LIN {X 0,Y 460.857,Z 363.08,A -85,B 0,C 180,E1 -7830,E2 -7830} C_VEL
LIN {X 0,Y 460.803,Z 363.083,A -85,B 0,C 180,E1 -7832.623,E2 -7832.623} C_VEL
LIN {X 0,Y 460.705,Z 363.097,A -85,B 0,C 180,E1 -7836.13,E2 -7836.13} C_VEL
LIN {X 0,Y 460.632,Z 363.107,A -85,B 0,C 180,E1 -7838.776,E2 -7838.776} C_VEL
LIN {X 0,Y 460.617,Z 363.108,A -85,B 0,C 180,E1 -7842.445,E2 -7842.445} C_VEL
LIN {X 0,Y 460.603,Z 363.11,A -85,B 0,C 180,E1 -7845.998,E2 -7845.998} C_VEL
LIN {X 0,Y 460.574,Z 363.115,A -85,B 0,C 180,E1 -7848.902,E2 -7848.902} C_VEL
LIN {X 0,Y 460.519,Z 363.121,A -85,B 0,C 180,E1 -7851.486,E2 -7851.486} C_VEL
LIN {X 0,Y 460.534,Z 363.116,A -85,B 0,C 180,E1 -7854.333,E2 -7854.333} C_VEL
LIN {X 0,Y 460.592,Z 363.111,A -85,B 0,C 180,E1 -7857.748,E2 -7857.748} C_VEL
LIN {X 0,Y 460.524,Z 363.12,A -85,B 0,C 180,E1 -7861.283,E2 -7861.283} C_VEL
LIN {X 0,Y 460.535,Z 363.117,A -85,B 0,C 180,E1 -7864.506,E2 -7864.506} C_VEL
LIN {X 0,Y 460.504,Z 363.122,A -85,B 0,C 180,E1 -7867.623,E2 -7867.623} C_VEL
LIN {X 0,Y 460.546,Z 363.118,A -85,B 0,C 180,E1 -7870.27,E2 -7870.27} C_VEL
LIN {X 0,Y 460.511,Z 363.123,A -85,B 0,C 180,E1 -7873.374,E2 -7873.374} C_VEL
LIN {X 0,Y 460.501,Z 363.121,A -85,B 0,C 180,E1 -7876.625,E2 -7876.625} C_VEL
LIN {X 0,Y 460.545,Z 363.117,A -85,B 0,C 180,E1 -7879.731,E2 -7879.731} C_VEL
LIN {X 0,Y 460.53,Z 363.121,A -85,B 0,C 180,E1 -7882.519,E2 -7882.519} C_VEL
LIN {X 0,Y 460.552,Z 363.117,A -85,B 0,C 180,E1 -7885.624,E2 -7885.624} C_VEL
LIN {X 0,Y 460.604,Z 363.114,A -85,B 0,C 180,E1 -7889.259,E2 -7889.259} C_VEL
LIN {X 0,Y 460.682,Z 363.307,A -85,B 0,C 180,E1 -7889.646,E2 -7889.646} C_VEL
LIN {X 0,Y 460.51,Z 369.483,A -85,B 0,C 180,E1 -7892.752,E2 -7892.752} C_VEL
LIN {X 0,Y 460.34,Z 375.322,A -85,B 0,C 180,E1 -7895.656,E2 -7895.656} C_VEL
LIN {X 0,Y 460.199,Z 381.499,A -85,B 0,C 180,E1 -7898.682,E2 -7898.682} C_VEL
LIN {X 0,Y 460.139,Z 386.881,A -85,B 0,C 180,E1 -7901.292,E2 -7901.292} C_VEL
LIN {X 0,Y 460.006,Z 394.526,A -85,B 0,C 180,E1 -7904.946,E2 -7904.946} C_VEL
LIN {X 0,Y 459.852,Z 402.194,A -85,B 0,C 180,E1 -7908.54,E2 -7908.54} C_VEL
LIN {X 0,Y 459.783,Z 406.743,A -85,B 0,C 180,E1 -7910.653,E2 -7910.653} C_VEL
LIN {X 0,Y 461.225,Z 417.498,A -85,B 0,C 180,E1 -7911.18,E2 -7911.18} C_VEL
LIN {X 0,Y 461.038,Z 426.889,A -85,B 0,C 180,E1 -7911.784,E2 -7911.784} C_VEL
LIN {X 0,Y 460.745,Z 435.524,A -85,B 0,C 180,E1 -7912.518,E2 -7912.518} C_VEL
LIN {X 0,Y 460.495,Z 443.706,A -85,B 0,C 180,E1 -7913.427,E2 -7913.427} C_VEL
LIN {X 0,Y 460.374,Z 451.186,A -85,B 0,C 180,E1 -7914.525,E2 -7914.525} C_VEL
LIN {X 0,Y 460.236,Z 456.815,A -85,B 0,C 180,E1 -7915.621,E2 -7915.621} C_VEL
LIN {X 0,Y 460.036,Z 461.668,A -85,B 0,C 180,E1 -7916.935,E2 -7916.935} C_VEL
LIN {X 0,Y 459.729,Z 464.779,A -85,B 0,C 180,E1 -7918.248,E2 -7918.248} C_VEL
LIN {X 0,Y 459.705,Z 465.955,A -85,B 0,C 180,E1 -7919.124,E2 -7919.124} C_VEL
LIN {X 0,Y 459.709,Z 466.457,A -85,B 0,C 180,E1 -7920,E2 -7920} C_VEL
LIN {X 0,Y 459.728,Z 466.292,A -85,B 0,C 180,E1 -7920.876,E2 -7920.876} C_VEL
LIN {X 0,Y 459.777,Z 465.459,A -85,B 0,C 180,E1 -7921.752,E2 -7921.752} C_VEL
LIN {X 0,Y 459.881,Z 463.94,A -85,B 0,C 180,E1 -7922.628,E2 -7922.628} C_VEL
LIN {X 0,Y 460.083,Z 461.69,A -85,B 0,C 180,E1 -7923.503,E2 -7923.503} C_VEL
LIN {X 0,Y 460.26,Z 458.652,A -85,B 0,C 180,E1 -7924.379,E2 -7924.379} C_VEL
LIN {X 0,Y 460.554,Z 453.616,A -85,B 0,C 180,E1 -7925.473,E2 -7925.473} C_VEL
LIN {X 0,Y 460.635,Z 448.398,A -85,B 0,C 180,E1 -7926.351,E2 -7926.351} C_VEL
LIN {X 0,Y 460.94,Z 441.818,A -85,B 0,C 180,E1 -7927.225,E2 -7927.225} C_VEL
LIN {X 0,Y 461.316,Z 433.586,A -85,B 0,C 180,E1 -7928.079,E2 -7928.079} C_VEL
LIN {X 0,Y 461.561,Z 425.177,A -85,B 0,C 180,E1 -7928.758,E2 -7928.758} C_VEL
LIN {X 0,Y 461.706,Z 418.277,A -85,B 0,C 180,E1 -7929.197,E2 -7929.197} C_VEL
LIN {X 0,Y 460.031,Z 408.765,A -85,B 0,C 180,E1 -7929.73,E2 -7929.73} C_VEL
LIN {X 0,Y 460.19,Z 403.416,A -85,B 0,C 180,E1 -7932.346,E2 -7932.346} C_VEL
LIN {X 0,Y 460.378,Z 396.222,A -85,B 0,C 180,E1 -7935.949,E2 -7935.949} C_VEL
LIN {X 0,Y 460.577,Z 390.465,A -85,B 0,C 180,E1 -7938.903,E2 -7938.903} C_VEL
LIN {X 0,Y 460.804,Z 383.745,A -85,B 0,C 180,E1 -7942.414,E2 -7942.414} C_VEL
LIN {X 0,Y 461.153,Z 377.222,A -85,B 0,C 180,E1 -7945.951,E2 -7945.951} C_VEL
LIN {X 0,Y 461.492,Z 371.525,A -85,B 0,C 180,E1 -7949.165,E2 -7949.165} C_VEL
LIN {X 0,Y 461.341,Z 367.729,A -85,B 0,C 180,E1 -7951.449,E2 -7951.449} C_VEL
LIN {X 0,Y 460.927,Z 364.949,A -85,B 0,C 180,E1 -7953.292,E2 -7953.292} C_VEL
LIN {X 0,Y 460.541,Z 363.122,A -85,B 0,C 180,E1 -7954.681,E2 -7954.681} C_VEL
LIN {X 0,Y 460.533,Z 363.122,A -85,B 0,C 180,E1 -7957.62,E2 -7957.62} C_VEL
LIN {X 0,Y 460.564,Z 363.118,A -85,B 0,C 180,E1 -7960.272,E2 -7960.272} C_VEL
LIN {X 0,Y 460.528,Z 363.122,A -85,B 0,C 180,E1 -7963.372,E2 -7963.372} C_VEL
LIN {X 0,Y 460.512,Z 363.124,A -85,B 0,C 180,E1 -7966.626,E2 -7966.626} C_VEL
LIN {X 0,Y 460.546,Z 363.121,A -85,B 0,C 180,E1 -7969.73,E2 -7969.73} C_VEL
LIN {X 0,Y 460.502,Z 363.126,A -85,B 0,C 180,E1 -7972.524,E2 -7972.524} C_VEL
LIN {X 0,Y 460.517,Z 363.332,A -85,B 0,C 180,E1 -7973.621,E2 -7973.621} C_VEL
LIN {X 0,Y 461.719,Z 367.784,A -85,B 0,C 180,E1 -7975.723,E2 -7975.723} C_VEL
LIN {X 0,Y 463.014,Z 373.479,A -85,B 0,C 180,E1 -7977.909,E2 -7977.909} C_VEL
LIN {X 0,Y 464.367,Z 379.853,A -85,B 0,C 180,E1 -7980.037,E2 -7980.037} C_VEL
LIN {X 0,Y 464.726,Z 384.238,A -85,B 0,C 180,E1 -7981.298,E2 -7981.298} C_VEL
LIN {X 0,Y 463.505,Z 394.628,A -85,B 0,C 180,E1 -7983.914,E2 -7983.914} C_VEL
LIN {X 0,Y 462.368,Z 407.715,A -85,B 0,C 180,E1 -7986.958,E2 -7986.958} C_VEL
LIN {X 0,Y 461.482,Z 422.533,A -85,B 0,C 180,E1 -7990.193,E2 -7990.193} C_VEL
LIN {X 0,Y 460.787,Z 438.027,A -85,B 0,C 180,E1 -7993.405,E2 -7993.405} C_VEL
LIN {X 0,Y 460.585,Z 444.606,A -85,B 0,C 180,E1 -7994.739,E2 -7994.739} C_VEL
LIN {X 0,Y 462.033,Z 459.219,A -85,B 0,C 180,E1 -7995.154,E2 -7995.154} C_VEL
LIN {X 0,Y 462.409,Z 464.775,A -85,B 0,C 180,E1 -7995.364,E2 -7995.364} C_VEL
LIN {X 0,Y 462.099,Z 476.978,A -85,B 0,C 180,E1 -7995.916,E2 -7995.916} C_VEL
LIN {X 0,Y 461.61,Z 489.57,A -85,B 0,C 180,E1 -7996.686,E2 -7996.686} C_VEL
LIN {X 0,Y 461.252,Z 500.147,A -85,B 0,C 180,E1 -7997.513,E2 -7997.513} C_VEL
LIN {X 0,Y 460.68,Z 509.899,A -85,B 0,C 180,E1 -7998.449,E2 -7998.449} C_VEL
LIN {X 0,Y 460.444,Z 518.389,A -85,B 0,C 180,E1 -7999.446,E2 -7999.446} C_VEL
LIN {X 0,Y 460.109,Z 527.598,A -85,B 0,C 180,E1 -8000.771,E2 -8000.771} C_VEL
LIN {X 0,Y 459.907,Z 535.009,A -85,B 0,C 180,E1 -8002.095,E2 -8002.095} C_VEL
LIN {X 0,Y 459.813,Z 541.057,A -85,B 0,C 180,E1 -8003.461,E2 -8003.461} C_VEL
LIN {X 0,Y 459.737,Z 545.498,A -85,B 0,C 180,E1 -8004.737,E2 -8004.737} C_VEL
LIN {X 0,Y 459.701,Z 547.925,A -85,B 0,C 180,E1 -8005.616,E2 -8005.616} C_VEL
LIN {X 0,Y 459.75,Z 549.915,A -85,B 0,C 180,E1 -8006.494,E2 -8006.494} C_VEL
LIN {X 0,Y 459.762,Z 551.424,A -85,B 0,C 180,E1 -8007.371,E2 -8007.371} C_VEL
LIN {X 0,Y 459.603,Z 553.141,A -85,B 0,C 180,E1 -8009.124,E2 -8009.124} C_VEL
LIN {X 0,Y 459.605,Z 553.392,A -85,B 0,C 180,E1 -8010,E2 -8010} C_VEL
LIN {X 0,Y 459.6,Z 553.186,A -85,B 0,C 180,E1 -8010.876,E2 -8010.876} C_VEL
LIN {X 0,Y 459.762,Z 551.579,A -85,B 0,C 180,E1 -8012.628,E2 -8012.628} C_VEL
LIN {X 0,Y 459.745,Z 550.107,A -85,B 0,C 180,E1 -8013.505,E2 -8013.505} C_VEL
LIN {X 0,Y 459.657,Z 547.047,A -85,B 0,C 180,E1 -8014.824,E2 -8014.824} C_VEL
LIN {X 0,Y 459.729,Z 542.895,A -85,B 0,C 180,E1 -8016.143,E2 -8016.143} C_VEL
LIN {X 0,Y 459.854,Z 537.524,A -85,B 0,C 180,E1 -8017.464,E2 -8017.464} C_VEL
LIN {X 0,Y 460.017,Z 530.749,A -85,B 0,C 180,E1 -8018.788,E2 -8018.788} C_VEL
LIN {X 0,Y 460.304,Z 522.289,A -85,B 0,C 180,E1 -8020.112,E2 -8020.112} C_VEL
LIN {X 0,Y 460.715,Z 513.529,A -85,B 0,C 180,E1 -8021.215,E2 -8021.215} C_VEL
LIN {X 0,Y 461.128,Z 503.892,A -85,B 0,C 180,E1 -8022.208,E2 -8022.208} C_VEL
LIN {X 0,Y 461.557,Z 493.026,A -85,B 0,C 180,E1 -8023.116,E2 -8023.116} C_VEL
LIN {X 0,Y 461.969,Z 481.615,A -85,B 0,C 180,E1 -8023.863,E2 -8023.863} C_VEL
LIN {X 0,Y 462.419,Z 468.145,A -85,B 0,C 180,E1 -8024.523,E2 -8024.523} C_VEL
LIN {X 0,Y 462.274,Z 461.426,A -85,B 0,C 180,E1 -8024.781,E2 -8024.781} C_VEL
LIN {X 0,Y 461.043,Z 449.191,A -85,B 0,C 180,E1 -8025.143,E2 -8025.143} C_VEL
LIN {X 0,Y 460.644,Z 445.197,A -85,B 0,C 180,E1 -8025.259,E2 -8025.259} C_VEL
LIN {X 0,Y 461.241,Z 428.609,A -85,B 0,C 180,E1 -8028.662,E2 -8028.662} C_VEL
LIN {X 0,Y 462.088,Z 413.087,A -85,B 0,C 180,E1 -8031.911,E2 -8031.911} C_VEL
LIN {X 0,Y 463.079,Z 396.786,A -85,B 0,C 180,E1 -8035.388,E2 -8035.388} C_VEL
LIN {X 0,Y 464.179,Z 382.26,A -85,B 0,C 180,E1 -8038.578,E2 -8038.578} C_VEL
LIN {X 0,Y 463.806,Z 378.299,A -85,B 0,C 180,E1 -8039.503,E2 -8039.503} C_VEL
LIN {X 0,Y 461.42,Z 367.379,A -85,B 0,C 180,E1 -8042.215,E2 -8042.215} C_VEL
LIN {X 0,Y 460.595,Z 363.115,A -85,B 0,C 180,E1 -8043.319,E2 -8043.319} C_VEL
LIN {X 0,Y 460.478,Z 363.127,A -85,B 0,C 180,E1 -8046.529,E2 -8046.529} C_VEL
LIN {X 0,Y 460.534,Z 363.12,A -85,B 0,C 180,E1 -8049.862,E2 -8049.862} C_VEL
LIN {X 0,Y 460.518,Z 363.121,A -85,B 0,C 180,E1 -8052.901,E2 -8052.901} C_VEL
LIN {X 0,Y 460.521,Z 363.121,A -85,B 0,C 180,E1 -8055.829,E2 -8055.829} C_VEL
LIN {X 0,Y 460.535,Z 363.117,A -85,B 0,C 180,E1 -8058.989,E2 -8058.989} C_VEL
LIN {X 0,Y 460.528,Z 363.118,A -85,B 0,C 180,E1 -8061.267,E2 -8061.267} C_VEL
LIN {X 0,Y 460.514,Z 363.121,A -85,B 0,C 180,E1 -8064.555,E2 -8064.555} C_VEL
LIN {X 0,Y 460.532,Z 363.119,A -85,B 0,C 180,E1 -8067.716,E2 -8067.716} C_VEL
LIN {X 0,Y 460.541,Z 363.116,A -85,B 0,C 180,E1 -8070.769,E2 -8070.769} C_VEL
LIN {X 0,Y 460.564,Z 363.118,A -85,B 0,C 180,E1 -8073.735,E2 -8073.735} C_VEL
LIN {X 0,Y 460.547,Z 363.119,A -85,B 0,C 180,E1 -8076.624,E2 -8076.624} C_VEL
LIN {X 0,Y 460.553,Z 363.116,A -85,B 0,C 180,E1 -8079.453,E2 -8079.453} C_VEL
LIN {X 0,Y 460.561,Z 363.115,A -85,B 0,C 180,E1 -8082.23,E2 -8082.23} C_VEL
LIN {X 0,Y 460.569,Z 363.114,A -85,B 0,C 180,E1 -8084.965,E2 -8084.965} C_VEL
LIN {X 0,Y 460.613,Z 363.11,A -85,B 0,C 180,E1 -8088.559,E2 -8088.559} C_VEL
LIN {X 0,Y 460.696,Z 363.099,A -85,B 0,C 180,E1 -8092.109,E2 -8092.109} C_VEL
LIN {X 0,Y 460.698,Z 363.097,A -85,B 0,C 180,E1 -8094.748,E2 -8094.748} C_VEL
LIN {X 0,Y 460.826,Z 363.083,A -85,B 0,C 180,E1 -8097.378,E2 -8097.378} C_VEL
LIN {X 0,Y 460.855,Z 363.081,A -85,B 0,C 180,E1 -8100,E2 -8100} C_VEL
LIN {X 0,Y 460.802,Z 363.084,A -85,B 0,C 180,E1 -8102.623,E2 -8102.623} C_VEL
LIN {X 0,Y 460.711,Z 363.095,A -85,B 0,C 180,E1 -8106.13,E2 -8106.13} C_VEL
LIN {X 0,Y 460.631,Z 363.109,A -85,B 0,C 180,E1 -8108.776,E2 -8108.776} C_VEL
LIN {X 0,Y 460.636,Z 363.106,A -85,B 0,C 180,E1 -8112.457,E2 -8112.457} C_VEL
LIN {X 0,Y 460.601,Z 363.108,A -85,B 0,C 180,E1 -8115.998,E2 -8115.998} C_VEL
LIN {X 0,Y 460.573,Z 363.116,A -85,B 0,C 180,E1 -8118.902,E2 -8118.902} C_VEL
LIN {X 0,Y 460.517,Z 363.122,A -85,B 0,C 180,E1 -8121.486,E2 -8121.486} C_VEL
LIN {X 0,Y 460.544,Z 363.116,A -85,B 0,C 180,E1 -8124.332,E2 -8124.332} C_VEL
LIN {X 0,Y 460.574,Z 363.115,A -85,B 0,C 180,E1 -8127.244,E2 -8127.244} C_VEL
LIN {X 0,Y 460.512,Z 363.122,A -85,B 0,C 180,E1 -8130.24,E2 -8130.24} C_VEL
LIN {X 0,Y 460.53,Z 363.122,A -85,B 0,C 180,E1 -8133.325,E2 -8133.325} C_VEL
LIN {X 0,Y 460.48,Z 363.125,A -85,B 0,C 180,E1 -8136.529,E2 -8136.529} C_VEL
LIN {X 0,Y 460.546,Z 363.119,A -85,B 0,C 180,E1 -8138.898,E2 -8138.898} C_VEL
LIN {X 0,Y 460.524,Z 363.122,A -85,B 0,C 180,E1 -8142.182,E2 -8142.182} C_VEL
LIN {X 0,Y 460.522,Z 363.121,A -85,B 0,C 180,E1 -8145.412,E2 -8145.412} C_VEL
LIN {X 0,Y 460.537,Z 363.119,A -85,B 0,C 180,E1 -8148.397,E2 -8148.397} C_VEL
LIN {X 0,Y 460.528,Z 363.119,A -85,B 0,C 180,E1 -8151.267,E2 -8151.267} C_VEL
LIN {X 0,Y 460.512,Z 363.122,A -85,B 0,C 180,E1 -8154.555,E2 -8154.555} C_VEL
LIN {X 0,Y 460.533,Z 363.118,A -85,B 0,C 180,E1 -8157.716,E2 -8157.716} C_VEL
LIN {X 0,Y 460.542,Z 363.118,A -85,B 0,C 180,E1 -8160.769,E2 -8160.769} C_VEL
LIN {X 0,Y 460.565,Z 363.116,A -85,B 0,C 180,E1 -8163.735,E2 -8163.735} C_VEL
LIN {X 0,Y 460.548,Z 363.119,A -85,B 0,C 180,E1 -8166.624,E2 -8166.624} C_VEL
LIN {X 0,Y 460.555,Z 363.114,A -85,B 0,C 180,E1 -8169.453,E2 -8169.453} C_VEL
LIN {X 0,Y 460.563,Z 363.118,A -85,B 0,C 180,E1 -8172.23,E2 -8172.23} C_VEL
LIN {X 0,Y 460.573,Z 363.115,A -85,B 0,C 180,E1 -8174.965,E2 -8174.965} C_VEL
LIN {X 0,Y 460.614,Z 363.112,A -85,B 0,C 180,E1 -8178.56,E2 -8178.56} C_VEL
LIN {X 0,Y 460.58,Z 363.112,A -85,B 0,C 180,E1 -8179.225,E2 -8179.225} C_VEL
LIN {X 0,Y 459.924,Z 363.197,A -85,B 0,C 180,E1 -8179.955,E2 -8179.955} C_VEL
LIN {X 0,Y 457.104,Z 363.545,A -85,B 0,C 180,E1 -8181.141,E2 -8181.141} C_VEL
LIN {X 0,Y 454.722,Z 363.846,A -85,B 0,C 180,E1 -8182.098,E2 -8182.098} C_VEL
LIN {X 0,Y 453.709,Z 363.968,A -85,B 0,C 180,E1 -8182.837,E2 -8182.837} C_VEL
LIN {X 0,Y 453.632,Z 363.977,A -85,B 0,C 180,E1 -8183.087,E2 -8183.087} C_VEL
LIN {X 0,Y 453.672,Z 363.973,A -85,B 0,C 180,E1 -8184.667,E2 -8184.667} C_VEL
LIN {X 0,Y 453.747,Z 363.965,A -85,B 0,C 180,E1 -8187.337,E2 -8187.337} C_VEL
LIN {X 0,Y 453.828,Z 363.955,A -85,B 0,C 180,E1 -8190,E2 -8190} C_VEL
LIN {X 0,Y 453.747,Z 363.962,A -85,B 0,C 180,E1 -8192.663,E2 -8192.663} C_VEL
LIN {X 0,Y 453.673,Z 363.973,A -85,B 0,C 180,E1 -8196.226,E2 -8196.226} C_VEL
LIN {X 0,Y 453.596,Z 363.984,A -85,B 0,C 180,E1 -8198.913,E2 -8198.913} C_VEL
LIN {X 0,Y 453.567,Z 363.985,A -85,B 0,C 180,E1 -8202.529,E2 -8202.529} C_VEL
LIN {X 0,Y 453.548,Z 363.988,A -85,B 0,C 180,E1 -8206.196,E2 -8206.196} C_VEL
LIN {X 0,Y 453.524,Z 363.994,A -85,B 0,C 180,E1 -8209.041,E2 -8209.041} C_VEL
LIN {X 0,Y 453.48,Z 364,A -85,B 0,C 180,E1 -8211.836,E2 -8211.836} C_VEL
LIN {X 0,Y 453.504,Z 363.992,A -85,B 0,C 180,E1 -8214.735,E2 -8214.735} C_VEL
LIN {X 0,Y 453.541,Z 363.99,A -85,B 0,C 180,E1 -8217.961,E2 -8217.961} C_VEL
LIN {X 0,Y 453.469,Z 363.999,A -85,B 0,C 180,E1 -8221.525,E2 -8221.525} C_VEL
LIN {X 0,Y 453.49,Z 363.995,A -85,B 0,C 180,E1 -8224.777,E2 -8224.777} C_VEL
LIN {X 0,Y 453.468,Z 363.999,A -85,B 0,C 180,E1 -8228.312,E2 -8228.312} C_VEL
LIN {X 0,Y 453.497,Z 363.996,A -85,B 0,C 180,E1 -8230.609,E2 -8230.609} C_VEL
LIN {X 0,Y 453.465,Z 364,A -85,B 0,C 180,E1 -8233.245,E2 -8233.245} C_VEL
LIN {X 0,Y 453.466,Z 363.999,A -85,B 0,C 180,E1 -8235.779,E2 -8235.779} C_VEL
LIN {X 0,Y 453.482,Z 363.996,A -85,B 0,C 180,E1 -8238.209,E2 -8238.209} C_VEL
LIN {X 0,Y 453.513,Z 363.996,A -85,B 0,C 180,E1 -8240.791,E2 -8240.791} C_VEL
LIN {X 0,Y 453.46,Z 364,A -85,B 0,C 180,E1 -8243.917,E2 -8243.917} C_VEL
LIN {X 0,Y 453.487,Z 364,A -85,B 0,C 180,E1 -8247.151,E2 -8247.151} C_VEL
LIN {X 0,Y 453.577,Z 364.027,A -85,B 0,C 180,E1 -8249.503,E2 -8249.503} C_VEL
LIN {X 0,Y 453.506,Z 369.486,A -85,B 0,C 180,E1 -8252.295,E2 -8252.295} C_VEL
LIN {X 0,Y 453.315,Z 375.395,A -85,B 0,C 180,E1 -8255.254,E2 -8255.254} C_VEL
LIN {X 0,Y 453.165,Z 381.948,A -85,B 0,C 180,E1 -8258.517,E2 -8258.517} C_VEL
LIN {X 0,Y 453.027,Z 388.938,A -85,B 0,C 180,E1 -8261.924,E2 -8261.924} C_VEL
LIN {X 0,Y 452.966,Z 394.742,A -85,B 0,C 180,E1 -8264.706,E2 -8264.706} C_VEL
LIN {X 0,Y 452.795,Z 402.443,A -85,B 0,C 180,E1 -8268.359,E2 -8268.359} C_VEL
LIN {X 0,Y 452.734,Z 407.048,A -85,B 0,C 180,E1 -8270.506,E2 -8270.506} C_VEL
LIN {X 0,Y 454.161,Z 416.831,A -85,B 0,C 180,E1 -8270.986,E2 -8270.986} C_VEL
LIN {X 0,Y 454.065,Z 425.727,A -85,B 0,C 180,E1 -8271.544,E2 -8271.544} C_VEL
LIN {X 0,Y 453.838,Z 433.911,A -85,B 0,C 180,E1 -8272.213,E2 -8272.213} C_VEL
LIN {X 0,Y 453.47,Z 442.344,A -85,B 0,C 180,E1 -8273.101,E2 -8273.101} C_VEL
LIN {X 0,Y 453.405,Z 448.927,A -85,B 0,C 180,E1 -8273.994,E2 -8273.994} C_VEL
LIN {X 0,Y 453.237,Z 455.281,A -85,B 0,C 180,E1 -8275.108,E2 -8275.108} C_VEL
LIN {X 0,Y 453.022,Z 460.828,A -85,B 0,C 180,E1 -8276.442,E2 -8276.442} C_VEL
LIN {X 0,Y 452.8,Z 463.498,A -85,B 0,C 180,E1 -8277.331,E2 -8277.331} C_VEL
LIN {X 0,Y 452.666,Z 465.412,A -85,B 0,C 180,E1 -8278.221,E2 -8278.221} C_VEL
LIN {X 0,Y 452.637,Z 466.617,A -85,B 0,C 180,E1 -8279.11,E2 -8279.11} C_VEL
LIN {X 0,Y 452.643,Z 467.146,A -85,B 0,C 180,E1 -8280,E2 -8280} C_VEL
LIN {X 0,Y 452.666,Z 467.006,A -85,B 0,C 180,E1 -8280.89,E2 -8280.89} C_VEL
LIN {X 0,Y 452.719,Z 466.196,A -85,B 0,C 180,E1 -8281.779,E2 -8281.779} C_VEL
LIN {X 0,Y 452.83,Z 464.701,A -85,B 0,C 180,E1 -8282.669,E2 -8282.669} C_VEL
LIN {X 0,Y 453.048,Z 462.476,A -85,B 0,C 180,E1 -8283.558,E2 -8283.558} C_VEL
LIN {X 0,Y 453.237,Z 459.477,A -85,B 0,C 180,E1 -8284.447,E2 -8284.447} C_VEL
LIN {X 0,Y 453.547,Z 454.511,A -85,B 0,C 180,E1 -8285.558,E2 -8285.558} C_VEL
LIN {X 0,Y 453.728,Z 447.9,A -85,B 0,C 180,E1 -8286.671,E2 -8286.671} C_VEL
LIN {X 0,Y 454.14,Z 440.066,A -85,B 0,C 180,E1 -8287.668,E2 -8287.668} C_VEL
LIN {X 0,Y 454.448,Z 432.198,A -85,B 0,C 180,E1 -8288.448,E2 -8288.448} C_VEL
LIN {X 0,Y 454.75,Z 423.545,A -85,B 0,C 180,E1 -8289.115,E2 -8289.115} C_VEL
LIN {X 0,Y 454.682,Z 418.192,A -85,B 0,C 180,E1 -8289.453,E2 -8289.453} C_VEL
LIN {X 0,Y 453.006,Z 409.211,A -85,B 0,C 180,E1 -8289.967,E2 -8289.967} C_VEL
LIN {X 0,Y 453.164,Z 404.055,A -85,B 0,C 180,E1 -8292.54,E2 -8292.54} C_VEL
LIN {X 0,Y 453.392,Z 396.849,A -85,B 0,C 180,E1 -8296.202,E2 -8296.202} C_VEL
LIN {X 0,Y 453.572,Z 391.35,A -85,B 0,C 180,E1 -8299.058,E2 -8299.058} C_VEL
LIN {X 0,Y 453.768,Z 386.166,A -85,B 0,C 180,E1 -8301.821,E2 -8301.821} C_VEL
LIN {X 0,Y 454.027,Z 380.917,A -85,B 0,C 180,E1 -8304.705,E2 -8304.705} C_VEL
LIN {X 0,Y 454.4,Z 375.73,A -85,B 0,C 180,E1 -8307.645,E2 -8307.645} C_VEL
LIN {X 0,Y 454.627,Z 371.692,A -85,B 0,C 180,E1 -8310.037,E2 -8310.037} C_VEL
LIN {X 0,Y 454.186,Z 367.518,A -85,B 0,C 180,E1 -8312.792,E2 -8312.792} C_VEL
LIN {X 0,Y 453.479,Z 364.001,A -85,B 0,C 180,E1 -8315.465,E2 -8315.465} C_VEL
LIN {X 0,Y 453.489,Z 364,A -85,B 0,C 180,E1 -8318.309,E2 -8318.309} C_VEL
LIN {X 0,Y 453.519,Z 363.995,A -85,B 0,C 180,E1 -8320.606,E2 -8320.606} C_VEL
LIN {X 0,Y 453.485,Z 363.999,A -85,B 0,C 180,E1 -8323.248,E2 -8323.248} C_VEL
LIN {X 0,Y 453.476,Z 364,A -85,B 0,C 180,E1 -8325.78,E2 -8325.78} C_VEL
LIN {X 0,Y 453.485,Z 364,A -85,B 0,C 180,E1 -8328.21,E2 -8328.21} C_VEL
LIN {X 0,Y 453.513,Z 363.996,A -85,B 0,C 180,E1 -8330.791,E2 -8330.791} C_VEL
LIN {X 0,Y 453.488,Z 364.196,A -85,B 0,C 180,E1 -8332.668,E2 -8332.668} C_VEL
LIN {X 0,Y 454.704,Z 368.932,A -85,B 0,C 180,E1 -8335.118,E2 -8335.118} C_VEL
LIN {X 0,Y 456.017,Z 374.334,A -85,B 0,C 180,E1 -8337.356,E2 -8337.356} C_VEL
LIN {X 0,Y 457.641,Z 382.209,A -85,B 0,C 180,E1 -8340.059,E2 -8340.059} C_VEL
LIN {X 0,Y 457.921,Z 385.915,A -85,B 0,C 180,E1 -8341.168,E2 -8341.168} C_VEL
LIN {X 0,Y 456.749,Z 394.867,A -85,B 0,C 180,E1 -8343.498,E2 -8343.498} C_VEL
LIN {X 0,Y 455.483,Z 407.713,A -85,B 0,C 180,E1 -8346.589,E2 -8346.589} C_VEL
LIN {X 0,Y 454.554,Z 422.357,A -85,B 0,C 180,E1 -8349.878,E2 -8349.878} C_VEL
LIN {X 0,Y 453.777,Z 437.577,A -85,B 0,C 180,E1 -8353.118,E2 -8353.118} C_VEL
LIN {X 0,Y 453.57,Z 444.565,A -85,B 0,C 180,E1 -8354.52,E2 -8354.52} C_VEL
LIN {X 0,Y 454.846,Z 457.367,A -85,B 0,C 180,E1 -8354.886,E2 -8354.886} C_VEL
LIN {X 0,Y 455.465,Z 465.322,A -85,B 0,C 180,E1 -8355.193,E2 -8355.193} C_VEL
LIN {X 0,Y 455.152,Z 476.153,A -85,B 0,C 180,E1 -8355.696,E2 -8355.696} C_VEL
LIN {X 0,Y 454.648,Z 488.774,A -85,B 0,C 180,E1 -8356.479,E2 -8356.479} C_VEL
LIN {X 0,Y 454.225,Z 500.002,A -85,B 0,C 180,E1 -8357.372,E2 -8357.372} C_VEL
LIN {X 0,Y 453.607,Z 510.137,A -85,B 0,C 180,E1 -8358.38,E2 -8358.38} C_VEL
LIN {X 0,Y 453.317,Z 519.313,A -85,B 0,C 180,E1 -8359.504,E2 -8359.504} C_VEL
LIN {X 0,Y 453.015,Z 528.254,A -85,B 0,C 180,E1 -8360.85,E2 -8360.85} C_VEL
LIN {X 0,Y 452.815,Z 535.355,A -85,B 0,C 180,E1 -8362.195,E2 -8362.195} C_VEL
LIN {X 0,Y 452.731,Z 540.774,A -85,B 0,C 180,E1 -8363.469,E2 -8363.469} C_VEL
LIN {X 0,Y 452.677,Z 544.812,A -85,B 0,C 180,E1 -8364.655,E2 -8364.655} C_VEL
LIN {X 0,Y 452.65,Z 548.3,A -85,B 0,C 180,E1 -8365.993,E2 -8365.993} C_VEL
LIN {X 0,Y 452.707,Z 550.755,A -85,B 0,C 180,E1 -8367.33,E2 -8367.33} C_VEL
LIN {X 0,Y 452.536,Z 552.476,A -85,B 0,C 180,E1 -8369.11,E2 -8369.11} C_VEL
LIN {X 0,Y 452.536,Z 552.725,A -85,B 0,C 180,E1 -8370,E2 -8370} C_VEL
LIN {X 0,Y 452.59,Z 551.909,A -85,B 0,C 180,E1 -8371.78,E2 -8371.78} C_VEL
LIN {X 0,Y 452.706,Z 550.904,A -85,B 0,C 180,E1 -8372.669,E2 -8372.669} C_VEL
LIN {X 0,Y 452.674,Z 549.416,A -85,B 0,C 180,E1 -8373.56,E2 -8373.56} C_VEL
LIN {X 0,Y 452.589,Z 546.337,A -85,B 0,C 180,E1 -8374.899,E2 -8374.899} C_VEL
LIN {X 0,Y 452.691,Z 541.261,A -85,B 0,C 180,E1 -8376.486,E2 -8376.486} C_VEL
LIN {X 0,Y 452.837,Z 534.667,A -85,B 0,C 180,E1 -8378.029,E2 -8378.029} C_VEL
LIN {X 0,Y 453.044,Z 527.293,A -85,B 0,C 180,E1 -8379.374,E2 -8379.374} C_VEL
LIN {X 0,Y 453.443,Z 518.107,A -85,B 0,C 180,E1 -8380.719,E2 -8380.719} C_VEL
LIN {X 0,Y 453.872,Z 507.418,A -85,B 0,C 180,E1 -8381.953,E2 -8381.953} C_VEL
LIN {X 0,Y 454.33,Z 496.566,A -85,B 0,C 180,E1 -8382.955,E2 -8382.955} C_VEL
LIN {X 0,Y 454.815,Z 485.74,A -85,B 0,C 180,E1 -8383.744,E2 -8383.744} C_VEL
LIN {X 0,Y 455.293,Z 472.8,A -85,B 0,C 180,E1 -8384.47,E2 -8384.47} C_VEL
LIN {X 0,Y 455.356,Z 462.669,A -85,B 0,C 180,E1 -8384.896,E2 -8384.896} C_VEL
LIN {X 0,Y 454.237,Z 450.854,A -85,B 0,C 180,E1 -8385.278,E2 -8385.278} C_VEL
LIN {X 0,Y 453.578,Z 444.953,A -85,B 0,C 180,E1 -8385.441,E2 -8385.441} C_VEL
LIN {X 0,Y 454.196,Z 429.258,A -85,B 0,C 180,E1 -8388.728,E2 -8388.728} C_VEL
LIN {X 0,Y 455.014,Z 415.009,A -85,B 0,C 180,E1 -8391.758,E2 -8391.758} C_VEL
LIN {X 0,Y 456.077,Z 398.702,A -85,B 0,C 180,E1 -8395.316,E2 -8395.316} C_VEL
LIN {X 0,Y 457.183,Z 384.551,A -85,B 0,C 180,E1 -8398.46,E2 -8398.46} C_VEL
LIN {X 0,Y 457.263,Z 381.851,A -85,B 0,C 180,E1 -8399.083,E2 -8399.083} C_VEL
LIN {X 0,Y 454.968,Z 370.857,A -85,B 0,C 180,E1 -8401.832,E2 -8401.832} C_VEL
LIN {X 0,Y 453.521,Z 363.995,A -85,B 0,C 180,E1 -8403.62,E2 -8403.62} C_VEL
LIN {X 0,Y 453.453,Z 364.001,A -85,B 0,C 180,E1 -8407.189,E2 -8407.189} C_VEL
LIN {X 0,Y 453.491,Z 363.995,A -85,B 0,C 180,E1 -8409.45,E2 -8409.45} C_VEL
LIN {X 0,Y 453.48,Z 364.001,A -85,B 0,C 180,E1 -8411.935,E2 -8411.935} C_VEL
LIN {X 0,Y 453.493,Z 363.997,A -85,B 0,C 180,E1 -8415.47,E2 -8415.47} C_VEL
LIN {X 0,Y 453.483,Z 363.999,A -85,B 0,C 180,E1 -8418.209,E2 -8418.209} C_VEL
LIN {X 0,Y 453.517,Z 363.991,A -85,B 0,C 180,E1 -8420.79,E2 -8420.79} C_VEL
LIN {X 0,Y 453.458,Z 364.002,A -85,B 0,C 180,E1 -8423.917,E2 -8423.917} C_VEL
LIN {X 0,Y 453.484,Z 363.997,A -85,B 0,C 180,E1 -8427.151,E2 -8427.151} C_VEL
LIN {X 0,Y 453.476,Z 364,A -85,B 0,C 180,E1 -8430.268,E2 -8430.268} C_VEL
LIN {X 0,Y 453.51,Z 363.993,A -85,B 0,C 180,E1 -8433.294,E2 -8433.294} C_VEL
LIN {X 0,Y 453.504,Z 363.995,A -85,B 0,C 180,E1 -8436.239,E2 -8436.239} C_VEL
LIN {X 0,Y 453.484,Z 363.997,A -85,B 0,C 180,E1 -8439.118,E2 -8439.118} C_VEL
LIN {X 0,Y 453.514,Z 363.996,A -85,B 0,C 180,E1 -8441.945,E2 -8441.945} C_VEL
LIN {X 0,Y 453.543,Z 363.989,A -85,B 0,C 180,E1 -8444.726,E2 -8444.726} C_VEL
LIN {X 0,Y 453.561,Z 363.989,A -85,B 0,C 180,E1 -8448.379,E2 -8448.379} C_VEL
LIN {X 0,Y 453.653,Z 363.977,A -85,B 0,C 180,E1 -8451.985,E2 -8451.985} C_VEL
LIN {X 0,Y 453.672,Z 363.972,A -85,B 0,C 180,E1 -8454.667,E2 -8454.667} C_VEL
LIN {X 0,Y 453.767,Z 363.963,A -85,B 0,C 180,E1 -8457.337,E2 -8457.337} C_VEL
LIN {X 0,Y 453.826,Z 363.957,A -85,B 0,C 180,E1 -8460,E2 -8460} C_VEL
LIN {X 0,Y 453.746,Z 363.963,A -85,B 0,C 180,E1 -8462.663,E2 -8462.663} C_VEL
LIN {X 0,Y 453.679,Z 363.971,A -85,B 0,C 180,E1 -8466.225,E2 -8466.225} C_VEL
LIN {X 0,Y 453.594,Z 363.986,A -85,B 0,C 180,E1 -8468.913,E2 -8468.913} C_VEL
LIN {X 0,Y 453.603,Z 363.982,A -85,B 0,C 180,E1 -8472.551,E2 -8472.551} C_VEL
LIN {X 0,Y 453.546,Z 363.987,A -85,B 0,C 180,E1 -8476.196,E2 -8476.196} C_VEL
LIN {X 0,Y 453.522,Z 363.994,A -85,B 0,C 180,E1 -8479.041,E2 -8479.041} C_VEL
LIN {X 0,Y 453.478,Z 363.999,A -85,B 0,C 180,E1 -8481.836,E2 -8481.836} C_VEL
LIN {X 0,Y 453.516,Z 363.993,A -85,B 0,C 180,E1 -8484.734,E2 -8484.734} C_VEL
LIN {X 0,Y 453.533,Z 363.989,A -85,B 0,C 180,E1 -8487.96,E2 -8487.96} C_VEL
LIN {X 0,Y 453.467,Z 364,A -85,B 0,C 180,E1 -8491.525,E2 -8491.525} C_VEL
LIN {X 0,Y 453.49,Z 363.997,A -85,B 0,C 180,E1 -8494.778,E2 -8494.778} C_VEL
LIN {X 0,Y 453.474,Z 363.997,A -85,B 0,C 180,E1 -8498.311,E2 -8498.311} C_VEL
LIN {X 0,Y 453.495,Z 363.998,A -85,B 0,C 180,E1 -8500.609,E2 -8500.609} C_VEL
LIN {X 0,Y 453.457,Z 364.002,A -85,B 0,C 180,E1 -8503.244,E2 -8503.244} C_VEL
LIN {X 0,Y 453.475,Z 363.998,A -85,B 0,C 180,E1 -8505.78,E2 -8505.78} C_VEL
LIN {X 0,Y 453.483,Z 363.996,A -85,B 0,C 180,E1 -8508.21,E2 -8508.21} C_VEL
LIN {X 0,Y 453.517,Z 363.993,A -85,B 0,C 180,E1 -8510.79,E2 -8510.79} C_VEL
LIN {X 0,Y 453.456,Z 364.002,A -85,B 0,C 180,E1 -8513.917,E2 -8513.917} C_VEL
LIN {X 0,Y 453.485,Z 363.997,A -85,B 0,C 180,E1 -8517.151,E2 -8517.151} C_VEL
LIN {X 0,Y 453.477,Z 364,A -85,B 0,C 180,E1 -8520.269,E2 -8520.269} C_VEL
LIN {X 0,Y 453.512,Z 363.994,A -85,B 0,C 180,E1 -8523.294,E2 -8523.294} C_VEL
LIN {X 0,Y 453.505,Z 363.994,A -85,B 0,C 180,E1 -8526.239,E2 -8526.239} C_VEL
LIN {X 0,Y 453.485,Z 363.996,A -85,B 0,C 180,E1 -8529.118,E2 -8529.118} C_VEL
LIN {X 0,Y 453.515,Z 363.994,A -85,B 0,C 180,E1 -8531.945,E2 -8531.945} C_VEL
LIN {X 0,Y 453.553,Z 363.989,A -85,B 0,C 180,E1 -8534.727,E2 -8534.727} C_VEL
LIN {X 0,Y 453.563,Z 363.989,A -85,B 0,C 180,E1 -8538.379,E2 -8538.379} C_VEL
LIN {X 0,Y 453.655,Z 363.978,A -85,B 0,C 180,E1 -8541.985,E2 -8541.985} C_VEL
LIN {X 0,Y 453.632,Z 363.977,A -85,B 0,C 180,E1 -8543.087,E2 -8543.087} C_VEL
LIN {X 0,Y 452.948,Z 364.067,A -85,B 0,C 180,E1 -8543.828,E2 -8543.828} C_VEL
LIN {X 0,Y 450.004,Z 364.43,A -85,B 0,C 180,E1 -8545.03,E2 -8545.03} C_VEL
LIN {X 0,Y 447.58,Z 364.733,A -85,B 0,C 180,E1 -8545.999,E2 -8545.999} C_VEL
LIN {X 0,Y 446.637,Z 364.851,A -85,B 0,C 180,E1 -8546.75,E2 -8546.75} C_VEL
LIN {X 0,Y 446.613,Z 364.852,A -85,B 0,C 180,E1 -8547.003,E2 -8547.003} C_VEL
LIN {X 0,Y 446.798,Z 364.831,A -85,B 0,C 180,E1 -8550,E2 -8550} C_VEL
LIN {X 0,Y 446.694,Z 364.84,A -85,B 0,C 180,E1 -8552.706,E2 -8552.706} C_VEL
LIN {X 0,Y 446.643,Z 364.849,A -85,B 0,C 180,E1 -8556.324,E2 -8556.324} C_VEL
LIN {X 0,Y 446.542,Z 364.862,A -85,B 0,C 180,E1 -8559.055,E2 -8559.055} C_VEL
LIN {X 0,Y 446.525,Z 364.862,A -85,B 0,C 180,E1 -8562.73,E2 -8562.73} C_VEL
LIN {X 0,Y 446.499,Z 364.866,A -85,B 0,C 180,E1 -8566.228,E2 -8566.228} C_VEL
LIN {X 0,Y 446.473,Z 364.871,A -85,B 0,C 180,E1 -8569.303,E2 -8569.303} C_VEL
LIN {X 0,Y 446.421,Z 364.877,A -85,B 0,C 180,E1 -8572.2,E2 -8572.2} C_VEL
LIN {X 0,Y 446.447,Z 364.873,A -85,B 0,C 180,E1 -8575.153,E2 -8575.153} C_VEL
LIN {X 0,Y 446.488,Z 364.869,A -85,B 0,C 180,E1 -8578.179,E2 -8578.179} C_VEL
LIN {X 0,Y 446.423,Z 364.879,A -85,B 0,C 180,E1 -8581.775,E2 -8581.775} C_VEL
LIN {X 0,Y 446.432,Z 364.874,A -85,B 0,C 180,E1 -8584.523,E2 -8584.523} C_VEL
LIN {X 0,Y 446.419,Z 364.876,A -85,B 0,C 180,E1 -8588.079,E2 -8588.079} C_VEL
LIN {X 0,Y 446.431,Z 364.877,A -85,B 0,C 180,E1 -8590.918,E2 -8590.918} C_VEL
LIN {X 0,Y 446.424,Z 364.877,A -85,B 0,C 180,E1 -8593.843,E2 -8593.843} C_VEL
LIN {X 0,Y 446.401,Z 364.877,A -85,B 0,C 180,E1 -8596.404,E2 -8596.404} C_VEL
LIN {X 0,Y 446.43,Z 364.878,A -85,B 0,C 180,E1 -8599.082,E2 -8599.082} C_VEL
LIN {X 0,Y 446.431,Z 364.876,A -85,B 0,C 180,E1 -8602.123,E2 -8602.123} C_VEL
LIN {X 0,Y 446.434,Z 364.877,A -85,B 0,C 180,E1 -8605.477,E2 -8605.477} C_VEL
LIN {X 0,Y 446.555,Z 364.864,A -85,B 0,C 180,E1 -8609.237,E2 -8609.237} C_VEL
LIN {X 0,Y 446.546,Z 365.007,A -85,B 0,C 180,E1 -8609.498,E2 -8609.498} C_VEL
LIN {X 0,Y 446.505,Z 369.5,A -85,B 0,C 180,E1 -8611.823,E2 -8611.823} C_VEL
LIN {X 0,Y 446.308,Z 375.434,A -85,B 0,C 180,E1 -8614.839,E2 -8614.839} C_VEL
LIN {X 0,Y 446.129,Z 382.443,A -85,B 0,C 180,E1 -8618.349,E2 -8618.349} C_VEL
LIN {X 0,Y 445.979,Z 389.11,A -85,B 0,C 180,E1 -8621.629,E2 -8621.629} C_VEL
LIN {X 0,Y 445.908,Z 394.912,A -85,B 0,C 180,E1 -8624.458,E2 -8624.458} C_VEL
LIN {X 0,Y 445.748,Z 402.682,A -85,B 0,C 180,E1 -8628.172,E2 -8628.172} C_VEL
LIN {X 0,Y 445.68,Z 407.431,A -85,B 0,C 180,E1 -8630.355,E2 -8630.355} C_VEL
LIN {X 0,Y 447.214,Z 418.235,A -85,B 0,C 180,E1 -8630.901,E2 -8630.901} C_VEL
LIN {X 0,Y 447.022,Z 427.638,A -85,B 0,C 180,E1 -8631.524,E2 -8631.524} C_VEL
LIN {X 0,Y 446.691,Z 437.09,A -85,B 0,C 180,E1 -8632.36,E2 -8632.36} C_VEL
LIN {X 0,Y 446.421,Z 444.683,A -85,B 0,C 180,E1 -8633.231,E2 -8633.231} C_VEL
LIN {X 0,Y 446.321,Z 452.163,A -85,B 0,C 180,E1 -8634.352,E2 -8634.352} C_VEL
LIN {X 0,Y 446.125,Z 457.889,A -85,B 0,C 180,E1 -8635.482,E2 -8635.482} C_VEL
LIN {X 0,Y 445.914,Z 462.842,A -85,B 0,C 180,E1 -8636.838,E2 -8636.838} C_VEL
LIN {X 0,Y 445.605,Z 466.044,A -85,B 0,C 180,E1 -8638.192,E2 -8638.192} C_VEL
LIN {X 0,Y 445.57,Z 467.278,A -85,B 0,C 180,E1 -8639.096,E2 -8639.096} C_VEL
LIN {X 0,Y 445.577,Z 467.836,A -85,B 0,C 180,E1 -8640,E2 -8640} C_VEL
LIN {X 0,Y 445.604,Z 467.726,A -85,B 0,C 180,E1 -8640.904,E2 -8640.904} C_VEL
LIN {X 0,Y 445.664,Z 466.95,A -85,B 0,C 180,E1 -8641.807,E2 -8641.807} C_VEL
LIN {X 0,Y 445.783,Z 465.494,A -85,B 0,C 180,E1 -8642.711,E2 -8642.711} C_VEL
LIN {X 0,Y 446.014,Z 463.316,A -85,B 0,C 180,E1 -8643.614,E2 -8643.614} C_VEL
LIN {X 0,Y 446.216,Z 460.368,A -85,B 0,C 180,E1 -8644.517,E2 -8644.517} C_VEL
LIN {X 0,Y 446.543,Z 455.461,A -85,B 0,C 180,E1 -8645.645,E2 -8645.645} C_VEL
LIN {X 0,Y 446.749,Z 448.944,A -85,B 0,C 180,E1 -8646.776,E2 -8646.776} C_VEL
LIN {X 0,Y 447.147,Z 442.106,A -85,B 0,C 180,E1 -8647.686,E2 -8647.686} C_VEL
LIN {X 0,Y 447.546,Z 433.522,A -85,B 0,C 180,E1 -8648.579,E2 -8648.579} C_VEL
LIN {X 0,Y 447.886,Z 423.456,A -85,B 0,C 180,E1 -8649.369,E2 -8649.369} C_VEL
LIN {X 0,Y 447.673,Z 418.153,A -85,B 0,C 180,E1 -8649.716,E2 -8649.716} C_VEL
LIN {X 0,Y 445.978,Z 409.708,A -85,B 0,C 180,E1 -8650.212,E2 -8650.212} C_VEL
LIN {X 0,Y 446.137,Z 404.693,A -85,B 0,C 180,E1 -8652.741,E2 -8652.741} C_VEL
LIN {X 0,Y 446.386,Z 397.494,A -85,B 0,C 180,E1 -8656.463,E2 -8656.463} C_VEL
LIN {X 0,Y 446.574,Z 392.135,A -85,B 0,C 180,E1 -8659.299,E2 -8659.299} C_VEL
LIN {X 0,Y 446.825,Z 386.854,A -85,B 0,C 180,E1 -8662.178,E2 -8662.178} C_VEL
LIN {X 0,Y 447.112,Z 381.624,A -85,B 0,C 180,E1 -8665.113,E2 -8665.113} C_VEL
LIN {X 0,Y 447.542,Z 376.523,A -85,B 0,C 180,E1 -8668.106,E2 -8668.106} C_VEL
LIN {X 0,Y 447.712,Z 372.946,A -85,B 0,C 180,E1 -8670.303,E2 -8670.303} C_VEL
LIN {X 0,Y 447.408,Z 370.07,A -85,B 0,C 180,E1 -8672.282,E2 -8672.282} C_VEL
LIN {X 0,Y 446.743,Z 366.323,A -85,B 0,C 180,E1 -8675.11,E2 -8675.11} C_VEL
LIN {X 0,Y 446.41,Z 364.881,A -85,B 0,C 180,E1 -8676.59,E2 -8676.59} C_VEL
LIN {X 0,Y 446.496,Z 364.87,A -85,B 0,C 180,E1 -8679.531,E2 -8679.531} C_VEL
LIN {X 0,Y 446.454,Z 364.876,A -85,B 0,C 180,E1 -8682.602,E2 -8682.602} C_VEL
LIN {X 0,Y 446.46,Z 364.874,A -85,B 0,C 180,E1 -8685.103,E2 -8685.103} C_VEL
LIN {X 0,Y 446.433,Z 364.878,A -85,B 0,C 180,E1 -8688.609,E2 -8688.609} C_VEL
LIN {X 0,Y 446.44,Z 365.004,A -85,B 0,C 180,E1 -8691.488,E2 -8691.488} C_VEL
LIN {X 0,Y 447.723,Z 370.15,A -85,B 0,C 180,E1 -8694.493,E2 -8694.493} C_VEL
LIN {X 0,Y 449.009,Z 375.257,A -85,B 0,C 180,E1 -8696.782,E2 -8696.782} C_VEL
LIN {X 0,Y 450.62,Z 382.977,A -85,B 0,C 180,E1 -8699.609,E2 -8699.609} C_VEL
LIN {X 0,Y 451.108,Z 386.62,A -85,B 0,C 180,E1 -8700.745,E2 -8700.745} C_VEL
LIN {X 0,Y 450.59,Z 391.465,A -85,B 0,C 180,E1 -8702.1,E2 -8702.1} C_VEL
LIN {X 0,Y 448.923,Z 405.173,A -85,B 0,C 180,E1 -8705.581,E2 -8705.581} C_VEL
LIN {X 0,Y 447.86,Z 418.05,A -85,B 0,C 180,E1 -8708.602,E2 -8708.602} C_VEL
LIN {X 0,Y 447.053,Z 431.861,A -85,B 0,C 180,E1 -8711.674,E2 -8711.674} C_VEL
LIN {X 0,Y 446.512,Z 443.969,A -85,B 0,C 180,E1 -8714.267,E2 -8714.267} C_VEL
LIN {X 0,Y 447.843,Z 456.24,A -85,B 0,C 180,E1 -8714.629,E2 -8714.629} C_VEL
LIN {X 0,Y 448.529,Z 466.005,A -85,B 0,C 180,E1 -8715.016,E2 -8715.016} C_VEL
LIN {X 0,Y 448.154,Z 477.455,A -85,B 0,C 180,E1 -8715.584,E2 -8715.584} C_VEL
LIN {X 0,Y 447.627,Z 489.649,A -85,B 0,C 180,E1 -8716.378,E2 -8716.378} C_VEL
LIN {X 0,Y 447.182,Z 500.557,A -85,B 0,C 180,E1 -8717.289,E2 -8717.289} C_VEL
LIN {X 0,Y 446.548,Z 511.43,A -85,B 0,C 180,E1 -8718.424,E2 -8718.424} C_VEL
LIN {X 0,Y 446.229,Z 520.284,A -85,B 0,C 180,E1 -8719.565,E2 -8719.565} C_VEL
LIN {X 0,Y 445.906,Z 528.836,A -85,B 0,C 180,E1 -8720.932,E2 -8720.932} C_VEL
LIN {X 0,Y 445.719,Z 535.71,A -85,B 0,C 180,E1 -8722.297,E2 -8722.297} C_VEL
LIN {X 0,Y 445.618,Z 541.19,A -85,B 0,C 180,E1 -8723.661,E2 -8723.661} C_VEL
LIN {X 0,Y 445.535,Z 545.433,A -85,B 0,C 180,E1 -8725.023,E2 -8725.023} C_VEL
LIN {X 0,Y 445.613,Z 548.576,A -85,B 0,C 180,E1 -8726.383,E2 -8726.383} C_VEL
LIN {X 0,Y 445.653,Z 550.09,A -85,B 0,C 180,E1 -8727.288,E2 -8727.288} C_VEL
LIN {X 0,Y 445.535,Z 551.15,A -85,B 0,C 180,E1 -8728.192,E2 -8728.192} C_VEL
LIN {X 0,Y 445.471,Z 551.81,A -85,B 0,C 180,E1 -8729.096,E2 -8729.096} C_VEL
LIN {X 0,Y 445.469,Z 552.053,A -85,B 0,C 180,E1 -8730,E2 -8730} C_VEL
LIN {X 0,Y 445.533,Z 551.231,A -85,B 0,C 180,E1 -8731.808,E2 -8731.808} C_VEL
LIN {X 0,Y 445.652,Z 550.22,A -85,B 0,C 180,E1 -8732.712,E2 -8732.712} C_VEL
LIN {X 0,Y 445.604,Z 548.714,A -85,B 0,C 180,E1 -8733.617,E2 -8733.617} C_VEL
LIN {X 0,Y 445.525,Z 545.614,A -85,B 0,C 180,E1 -8734.977,E2 -8734.977} C_VEL
LIN {X 0,Y 445.627,Z 540.842,A -85,B 0,C 180,E1 -8736.496,E2 -8736.496} C_VEL
LIN {X 0,Y 445.728,Z 534.943,A -85,B 0,C 180,E1 -8737.93,E2 -8737.93} C_VEL
LIN {X 0,Y 445.946,Z 527.802,A -85,B 0,C 180,E1 -8739.296,E2 -8739.296} C_VEL
LIN {X 0,Y 446.309,Z 518.835,A -85,B 0,C 180,E1 -8740.663,E2 -8740.663} C_VEL
LIN {X 0,Y 446.645,Z 509.579,A -85,B 0,C 180,E1 -8741.803,E2 -8741.803} C_VEL
LIN {X 0,Y 447.123,Z 500.536,A -85,B 0,C 180,E1 -8742.712,E2 -8742.712} C_VEL
LIN {X 0,Y 447.663,Z 489.327,A -85,B 0,C 180,E1 -8743.62,E2 -8743.62} C_VEL
LIN {X 0,Y 448.05,Z 478.705,A -85,B 0,C 180,E1 -8744.303,E2 -8744.303} C_VEL
LIN {X 0,Y 448.512,Z 465.891,A -85,B 0,C 180,E1 -8744.926,E2 -8744.926} C_VEL
LIN {X 0,Y 447.346,Z 452.424,A -85,B 0,C 180,E1 -8745.403,E2 -8745.403} C_VEL
LIN {X 0,Y 446.495,Z 444.695,A -85,B 0,C 180,E1 -8745.616,E2 -8745.616} C_VEL
LIN {X 0,Y 447.145,Z 429.868,A -85,B 0,C 180,E1 -8748.796,E2 -8748.796} C_VEL
LIN {X 0,Y 448.016,Z 415.726,A -85,B 0,C 180,E1 -8751.874,E2 -8751.874} C_VEL
LIN {X 0,Y 449.126,Z 399.397,A -85,B 0,C 180,E1 -8755.488,E2 -8755.488} C_VEL
LIN {X 0,Y 450.311,Z 385.385,A -85,B 0,C 180,E1 -8758.68,E2 -8758.68} C_VEL
LIN {X 0,Y 450.105,Z 382.066,A -85,B 0,C 180,E1 -8759.475,E2 -8759.475} C_VEL
LIN {X 0,Y 447.93,Z 371.845,A -85,B 0,C 180,E1 -8762.085,E2 -8762.085} C_VEL
LIN {X 0,Y 446.483,Z 364.872,A -85,B 0,C 180,E1 -8763.972,E2 -8763.972} C_VEL
LIN {X 0,Y 446.403,Z 364.881,A -85,B 0,C 180,E1 -8766.745,E2 -8766.745} C_VEL
LIN {X 0,Y 446.445,Z 364.877,A -85,B 0,C 180,E1 -8770.198,E2 -8770.198} C_VEL
LIN {X 0,Y 446.422,Z 364.878,A -85,B 0,C 180,E1 -8773.599,E2 -8773.599} C_VEL
LIN {X 0,Y 446.422,Z 364.878,A -85,B 0,C 180,E1 -8776.4,E2 -8776.4} C_VEL
LIN {X 0,Y 446.452,Z 364.873,A -85,B 0,C 180,E1 -8779.803,E2 -8779.803} C_VEL
LIN {X 0,Y 446.429,Z 364.878,A -85,B 0,C 180,E1 -8782.123,E2 -8782.123} C_VEL
LIN {X 0,Y 446.432,Z 364.877,A -85,B 0,C 180,E1 -8785.477,E2 -8785.477} C_VEL
LIN {X 0,Y 446.417,Z 364.877,A -85,B 0,C 180,E1 -8788.7,E2 -8788.7} C_VEL
LIN {X 0,Y 446.485,Z 364.871,A -85,B 0,C 180,E1 -8791.821,E2 -8791.821} C_VEL
LIN {X 0,Y 446.458,Z 364.872,A -85,B 0,C 180,E1 -8794.848,E2 -8794.848} C_VEL
LIN {X 0,Y 446.449,Z 364.876,A -85,B 0,C 180,E1 -8798.245,E2 -8798.245} C_VEL
LIN {X 0,Y 446.459,Z 364.873,A -85,B 0,C 180,E1 -8801.649,E2 -8801.649} C_VEL
LIN {X 0,Y 446.51,Z 364.865,A -85,B 0,C 180,E1 -8804.48,E2 -8804.48} C_VEL
LIN {X 0,Y 446.519,Z 364.867,A -85,B 0,C 180,E1 -8808.193,E2 -8808.193} C_VEL
LIN {X 0,Y 446.602,Z 364.857,A -85,B 0,C 180,E1 -8811.858,E2 -8811.858} C_VEL
LIN {X 0,Y 446.647,Z 364.847,A -85,B 0,C 180,E1 -8814.583,E2 -8814.583} C_VEL
LIN {X 0,Y 446.711,Z 364.843,A -85,B 0,C 180,E1 -8817.295,E2 -8817.295} C_VEL
LIN {X 0,Y 446.796,Z 364.832,A -85,B 0,C 180,E1 -8820,E2 -8820} C_VEL
LIN {X 0,Y 446.693,Z 364.842,A -85,B 0,C 180,E1 -8822.705,E2 -8822.705} C_VEL
LIN {X 0,Y 446.648,Z 364.847,A -85,B 0,C 180,E1 -8826.324,E2 -8826.324} C_VEL
LIN {X 0,Y 446.54,Z 364.863,A -85,B 0,C 180,E1 -8829.055,E2 -8829.055} C_VEL
LIN {X 0,Y 446.535,Z 364.862,A -85,B 0,C 180,E1 -8832.729,E2 -8832.729} C_VEL
LIN {X 0,Y 446.491,Z 364.866,A -85,B 0,C 180,E1 -8836.459,E2 -8836.459} C_VEL
LIN {X 0,Y 446.471,Z 364.871,A -85,B 0,C 180,E1 -8839.303,E2 -8839.303} C_VEL
LIN {X 0,Y 446.42,Z 364.877,A -85,B 0,C 180,E1 -8842.2,E2 -8842.2} C_VEL
LIN {X 0,Y 446.46,Z 364.875,A -85,B 0,C 180,E1 -8845.152,E2 -8845.152} C_VEL
LIN {X 0,Y 446.486,Z 364.868,A -85,B 0,C 180,E1 -8848.179,E2 -8848.179} C_VEL
LIN {X 0,Y 446.421,Z 364.878,A -85,B 0,C 180,E1 -8851.775,E2 -8851.775} C_VEL
LIN {X 0,Y 446.431,Z 364.875,A -85,B 0,C 180,E1 -8854.523,E2 -8854.523} C_VEL
LIN {X 0,Y 446.432,Z 364.873,A -85,B 0,C 180,E1 -8858.082,E2 -8858.082} C_VEL
LIN {X 0,Y 446.428,Z 364.876,A -85,B 0,C 180,E1 -8860.918,E2 -8860.918} C_VEL
LIN {X 0,Y 446.403,Z 364.879,A -85,B 0,C 180,E1 -8863.846,E2 -8863.846} C_VEL
LIN {X 0,Y 446.422,Z 364.876,A -85,B 0,C 180,E1 -8866.401,E2 -8866.401} C_VEL
LIN {X 0,Y 446.453,Z 364.871,A -85,B 0,C 180,E1 -8869.803,E2 -8869.803} C_VEL
LIN {X 0,Y 446.411,Z 364.88,A -85,B 0,C 180,E1 -8872.122,E2 -8872.122} C_VEL
LIN {X 0,Y 446.43,Z 364.876,A -85,B 0,C 180,E1 -8875.477,E2 -8875.477} C_VEL
LIN {X 0,Y 446.418,Z 364.88,A -85,B 0,C 180,E1 -8878.7,E2 -8878.7} C_VEL
LIN {X 0,Y 446.486,Z 364.869,A -85,B 0,C 180,E1 -8881.822,E2 -8881.822} C_VEL
LIN {X 0,Y 446.46,Z 364.873,A -85,B 0,C 180,E1 -8884.848,E2 -8884.848} C_VEL
LIN {X 0,Y 446.45,Z 364.874,A -85,B 0,C 180,E1 -8888.245,E2 -8888.245} C_VEL
LIN {X 0,Y 446.461,Z 364.871,A -85,B 0,C 180,E1 -8891.649,E2 -8891.649} C_VEL
LIN {X 0,Y 446.519,Z 364.865,A -85,B 0,C 180,E1 -8894.48,E2 -8894.48} C_VEL
LIN {X 0,Y 446.521,Z 364.865,A -85,B 0,C 180,E1 -8898.193,E2 -8898.193} C_VEL
LIN {X 0,Y 446.603,Z 364.855,A -85,B 0,C 180,E1 -8901.858,E2 -8901.858} C_VEL
LIN {X 0,Y 446.646,Z 364.848,A -85,B 0,C 180,E1 -8904.583,E2 -8904.583} C_VEL
LIN {X 0,Y 446.613,Z 364.852,A -85,B 0,C 180,E1 -8907.003,E2 -8907.003} C_VEL
LIN {X 0,Y 446.089,Z 364.92,A -85,B 0,C 180,E1 -8907.756,E2 -8907.756} C_VEL
LIN {X 0,Y 443.279,Z 365.271,A -85,B 0,C 180,E1 -8908.98,E2 -8908.98} C_VEL
LIN {X 0,Y 440.803,Z 365.578,A -85,B 0,C 180,E1 -8909.967,E2 -8909.967} C_VEL
LIN {X 0,Y 439.719,Z 365.711,A -85,B 0,C 180,E1 -8910.73,E2 -8910.73} C_VEL
LIN {X 0,Y 439.625,Z 365.722,A -85,B 0,C 180,E1 -8910.989,E2 -8910.989} C_VEL
LIN {X 0,Y 439.644,Z 365.718,A -85,B 0,C 180,E1 -8912.749,E2 -8912.749} C_VEL
LIN {X 0,Y 439.615,Z 365.725,A -85,B 0,C 180,E1 -8916.425,E2 -8916.425} C_VEL
LIN {X 0,Y 439.503,Z 365.74,A -85,B 0,C 180,E1 -8919.202,E2 -8919.202} C_VEL
LIN {X 0,Y 439.469,Z 365.741,A -85,B 0,C 180,E1 -8922.938,E2 -8922.938} C_VEL
LIN {X 0,Y 439.451,Z 365.745,A -85,B 0,C 180,E1 -8926.349,E2 -8926.349} C_VEL
LIN {X 0,Y 439.406,Z 365.751,A -85,B 0,C 180,E1 -8929.626,E2 -8929.626} C_VEL
LIN {X 0,Y 439.367,Z 365.754,A -85,B 0,C 180,E1 -8932.576,E2 -8932.576} C_VEL
LIN {X 0,Y 439.401,Z 365.754,A -85,B 0,C 180,E1 -8935.585,E2 -8935.585} C_VEL
LIN {X 0,Y 439.421,Z 365.749,A -85,B 0,C 180,E1 -8938.673,E2 -8938.673} C_VEL
LIN {X 0,Y 439.374,Z 365.756,A -85,B 0,C 180,E1 -8942.031,E2 -8942.031} C_VEL
LIN {X 0,Y 439.397,Z 365.754,A -85,B 0,C 180,E1 -8945.34,E2 -8945.34} C_VEL
LIN {X 0,Y 439.386,Z 365.753,A -85,B 0,C 180,E1 -8948.595,E2 -8948.595} C_VEL
LIN {X 0,Y 439.393,Z 365.753,A -85,B 0,C 180,E1 -8951.257,E2 -8951.257} C_VEL
LIN {X 0,Y 439.407,Z 365.75,A -85,B 0,C 180,E1 -8954.729,E2 -8954.729} C_VEL
LIN {X 0,Y 439.399,Z 365.75,A -85,B 0,C 180,E1 -8957.796,E2 -8957.796} C_VEL
LIN {X 0,Y 439.433,Z 365.747,A -85,B 0,C 180,E1 -8960.228,E2 -8960.228} C_VEL
LIN {X 0,Y 439.38,Z 365.755,A -85,B 0,C 180,E1 -8963.713,E2 -8963.713} C_VEL
LIN {X 0,Y 439.385,Z 365.756,A -85,B 0,C 180,E1 -8967.055,E2 -8967.055} C_VEL
LIN {X 0,Y 439.52,Z 365.858,A -85,B 0,C 180,E1 -8969.429,E2 -8969.429} C_VEL
LIN {X 0,Y 439.488,Z 369.978,A -85,B 0,C 180,E1 -8971.586,E2 -8971.586} C_VEL
LIN {X 0,Y 439.266,Z 375.481,A -85,B 0,C 180,E1 -8974.406,E2 -8974.406} C_VEL
LIN {X 0,Y 439.082,Z 381.4,A -85,B 0,C 180,E1 -8977.409,E2 -8977.409} C_VEL
LIN {X 0,Y 438.972,Z 388.248,A -85,B 0,C 180,E1 -8980.84,E2 -8980.84} C_VEL
LIN {X 0,Y 438.859,Z 395.106,A -85,B 0,C 180,E1 -8984.202,E2 -8984.202} C_VEL
LIN {X 0,Y 438.704,Z 402.923,A -85,B 0,C 180,E1 -8987.98,E2 -8987.98} C_VEL
LIN {X 0,Y 438.606,Z 407.759,A -85,B 0,C 180,E1 -8990.198,E2 -8990.198} C_VEL
LIN {X 0,Y 440.192,Z 418.596,A -85,B 0,C 180,E1 -8990.755,E2 -8990.755} C_VEL
LIN {X 0,Y 440.032,Z 427.99,A -85,B 0,C 180,E1 -8991.388,E2 -8991.388} C_VEL
LIN {X 0,Y 439.677,Z 437.466,A -85,B 0,C 180,E1 -8992.237,E2 -8992.237} C_VEL
LIN {X 0,Y 439.378,Z 445.389,A -85,B 0,C 180,E1 -8993.163,E2 -8993.163} C_VEL
LIN {X 0,Y 439.296,Z 452.617,A -85,B 0,C 180,E1 -8994.261,E2 -8994.261} C_VEL
LIN {X 0,Y 439.073,Z 458.39,A -85,B 0,C 180,E1 -8995.41,E2 -8995.41} C_VEL
LIN {X 0,Y 438.86,Z 463.392,A -85,B 0,C 180,E1 -8996.787,E2 -8996.787} C_VEL
LIN {X 0,Y 438.546,Z 466.654,A -85,B 0,C 180,E1 -8998.163,E2 -8998.163} C_VEL
LIN {X 0,Y 438.501,Z 467.93,A -85,B 0,C 180,E1 -8999.082,E2 -8999.082} C_VEL
LIN {X 0,Y 438.512,Z 468.527,A -85,B 0,C 180,E1 -9000,E2 -9000} C_VEL
LIN {X 0,Y 438.543,Z 468.455,A -85,B 0,C 180,E1 -9000.918,E2 -9000.918} C_VEL
LIN {X 0,Y 438.609,Z 467.714,A -85,B 0,C 180,E1 -9001.836,E2 -9001.836} C_VEL
LIN {X 0,Y 438.737,Z 466.294,A -85,B 0,C 180,E1 -9002.754,E2 -9002.754} C_VEL
LIN {X 0,Y 438.981,Z 464.154,A -85,B 0,C 180,E1 -9003.672,E2 -9003.672} C_VEL
LIN {X 0,Y 439.197,Z 461.253,A -85,B 0,C 180,E1 -9004.589,E2 -9004.589} C_VEL
LIN {X 0,Y 439.541,Z 456.4,A -85,B 0,C 180,E1 -9005.735,E2 -9005.735} C_VEL
LIN {X 0,Y 439.775,Z 449.991,A -85,B 0,C 180,E1 -9006.884,E2 -9006.884} C_VEL
LIN {X 0,Y 440.23,Z 442.97,A -85,B 0,C 180,E1 -9007.848,E2 -9007.848} C_VEL
LIN {X 0,Y 440.646,Z 434.938,A -85,B 0,C 180,E1 -9008.714,E2 -9008.714} C_VEL
LIN {X 0,Y 441.033,Z 425.308,A -85,B 0,C 180,E1 -9009.516,E2 -9009.516} C_VEL
LIN {X 0,Y 440.944,Z 420.173,A -85,B 0,C 180,E1 -9009.866,E2 -9009.866} C_VEL
LIN {X 0,Y 438.943,Z 410.144,A -85,B 0,C 180,E1 -9010.494,E2 -9010.494} C_VEL
LIN {X 0,Y 439.128,Z 405.372,A -85,B 0,C 180,E1 -9012.948,E2 -9012.948} C_VEL
LIN {X 0,Y 439.377,Z 398.947,A -85,B 0,C 180,E1 -9016.316,E2 -9016.316} C_VEL
LIN {X 0,Y 439.614,Z 392.837,A -85,B 0,C 180,E1 -9019.617,E2 -9019.617} C_VEL
LIN {X 0,Y 439.88,Z 387.596,A -85,B 0,C 180,E1 -9022.548,E2 -9022.548} C_VEL
LIN {X 0,Y 440.214,Z 382.423,A -85,B 0,C 180,E1 -9025.535,E2 -9025.535} C_VEL
LIN {X 0,Y 440.684,Z 377.183,A -85,B 0,C 180,E1 -9028.7,E2 -9028.7} C_VEL
LIN {X 0,Y 440.778,Z 374.175,A -85,B 0,C 180,E1 -9030.679,E2 -9030.679} C_VEL
LIN {X 0,Y 440.42,Z 371.122,A -85,B 0,C 180,E1 -9032.858,E2 -9032.858} C_VEL
LIN {X 0,Y 439.844,Z 367.993,A -85,B 0,C 180,E1 -9035.422,E2 -9035.422} C_VEL
LIN {X 0,Y 439.401,Z 365.754,A -85,B 0,C 180,E1 -9037.719,E2 -9037.719} C_VEL
LIN {X 0,Y 439.432,Z 365.75,A -85,B 0,C 180,E1 -9039.853,E2 -9039.853} C_VEL
LIN {X 0,Y 439.407,Z 365.754,A -85,B 0,C 180,E1 -9042.63,E2 -9042.63} C_VEL
LIN {X 0,Y 439.41,Z 365.753,A -85,B 0,C 180,E1 -9045.271,E2 -9045.271} C_VEL
LIN {X 0,Y 439.393,Z 365.755,A -85,B 0,C 180,E1 -9048.743,E2 -9048.743} C_VEL
LIN {X 0,Y 439.434,Z 365.936,A -85,B 0,C 180,E1 -9050.146,E2 -9050.146} C_VEL
LIN {X 0,Y 440.228,Z 369.393,A -85,B 0,C 180,E1 -9052.652,E2 -9052.652} C_VEL
LIN {X 0,Y 441.356,Z 373.725,A -85,B 0,C 180,E1 -9055.022,E2 -9055.022} C_VEL
LIN {X 0,Y 442.634,Z 379.005,A -85,B 0,C 180,E1 -9057.327,E2 -9057.327} C_VEL
LIN {X 0,Y 444.138,Z 386.68,A -85,B 0,C 180,E1 -9060.094,E2 -9060.094} C_VEL
LIN {X 0,Y 444.195,Z 390.124,A -85,B 0,C 180,E1 -9061.147,E2 -9061.147} C_VEL
LIN {X 0,Y 442.592,Z 401.111,A -85,B 0,C 180,E1 -9064.108,E2 -9064.108} C_VEL
LIN {X 0,Y 441.408,Z 412.934,A -85,B 0,C 180,E1 -9067.041,E2 -9067.041} C_VEL
LIN {X 0,Y 440.304,Z 427.39,A -85,B 0,C 180,E1 -9070.415,E2 -9070.415} C_VEL
LIN {X 0,Y 439.588,Z 441.728,A -85,B 0,C 180,E1 -9073.59,E2 -9073.59} C_VEL
LIN {X 0,Y 439.514,Z 443.875,A -85,B 0,C 180,E1 -9074.011,E2 -9074.011} C_VEL
LIN {X 0,Y 440.823,Z 455.387,A -85,B 0,C 180,E1 -9074.363,E2 -9074.363} C_VEL
LIN {X 0,Y 441.627,Z 466.761,A -85,B 0,C 180,E1 -9074.836,E2 -9074.836} C_VEL
LIN {X 0,Y 441.18,Z 478.842,A -85,B 0,C 180,E1 -9075.469,E2 -9075.469} C_VEL
LIN {X 0,Y 440.607,Z 490.508,A -85,B 0,C 180,E1 -9076.271,E2 -9076.271} C_VEL
LIN {X 0,Y 440.14,Z 501.114,A -85,B 0,C 180,E1 -9077.2,E2 -9077.2} C_VEL
LIN {X 0,Y 439.533,Z 510.793,A -85,B 0,C 180,E1 -9078.237,E2 -9078.237} C_VEL
LIN {X 0,Y 439.179,Z 519.633,A -85,B 0,C 180,E1 -9079.395,E2 -9079.395} C_VEL
LIN {X 0,Y 438.829,Z 528.175,A -85,B 0,C 180,E1 -9080.784,E2 -9080.784} C_VEL
LIN {X 0,Y 438.648,Z 535.056,A -85,B 0,C 180,E1 -9082.173,E2 -9082.173} C_VEL
LIN {X 0,Y 438.546,Z 540.535,A -85,B 0,C 180,E1 -9083.559,E2 -9083.559} C_VEL
LIN {X 0,Y 438.474,Z 544.777,A -85,B 0,C 180,E1 -9084.942,E2 -9084.942} C_VEL
LIN {X 0,Y 438.55,Z 547.918,A -85,B 0,C 180,E1 -9086.325,E2 -9086.325} C_VEL
LIN {X 0,Y 438.583,Z 549.426,A -85,B 0,C 180,E1 -9087.244,E2 -9087.244} C_VEL
LIN {X 0,Y 438.48,Z 550.487,A -85,B 0,C 180,E1 -9088.163,E2 -9088.163} C_VEL
LIN {X 0,Y 438.408,Z 551.144,A -85,B 0,C 180,E1 -9089.081,E2 -9089.081} C_VEL
LIN {X 0,Y 438.403,Z 551.375,A -85,B 0,C 180,E1 -9090,E2 -9090} C_VEL
LIN {X 0,Y 438.477,Z 550.542,A -85,B 0,C 180,E1 -9091.837,E2 -9091.837} C_VEL
LIN {X 0,Y 438.599,Z 549.519,A -85,B 0,C 180,E1 -9092.755,E2 -9092.755} C_VEL
LIN {X 0,Y 438.536,Z 547.993,A -85,B 0,C 180,E1 -9093.675,E2 -9093.675} C_VEL
LIN {X 0,Y 438.463,Z 544.866,A -85,B 0,C 180,E1 -9095.057,E2 -9095.057} C_VEL
LIN {X 0,Y 438.546,Z 540.464,A -85,B 0,C 180,E1 -9096.488,E2 -9096.488} C_VEL
LIN {X 0,Y 438.67,Z 534.123,A -85,B 0,C 180,E1 -9098.058,E2 -9098.058} C_VEL
LIN {X 0,Y 438.879,Z 526.905,A -85,B 0,C 180,E1 -9099.447,E2 -9099.447} C_VEL
LIN {X 0,Y 439.279,Z 517.878,A -85,B 0,C 180,E1 -9100.835,E2 -9100.835} C_VEL
LIN {X 0,Y 439.671,Z 508.507,A -85,B 0,C 180,E1 -9101.993,E2 -9101.993} C_VEL
LIN {X 0,Y 440.054,Z 499.317,A -85,B 0,C 180,E1 -9102.92,E2 -9102.92} C_VEL
LIN {X 0,Y 440.707,Z 487.971,A -85,B 0,C 180,E1 -9103.84,E2 -9103.84} C_VEL
LIN {X 0,Y 441.161,Z 476.117,A -85,B 0,C 180,E1 -9104.59,E2 -9104.59} C_VEL
LIN {X 0,Y 441.392,Z 464.439,A -85,B 0,C 180,E1 -9105.143,E2 -9105.143} C_VEL
LIN {X 0,Y 440.224,Z 451.554,A -85,B 0,C 180,E1 -9105.599,E2 -9105.599} C_VEL
LIN {X 0,Y 439.44,Z 444.603,A -85,B 0,C 180,E1 -9105.776,E2 -9105.776} C_VEL
LIN {X 0,Y 440.091,Z 430.432,A -85,B 0,C 180,E1 -9108.867,E2 -9108.867} C_VEL
LIN {X 0,Y 440.921,Z 417.425,A -85,B 0,C 180,E1 -9111.752,E2 -9111.752} C_VEL
LIN {X 0,Y 441.962,Z 403.128,A -85,B 0,C 180,E1 -9114.986,E2 -9114.986} C_VEL
LIN {X 0,Y 443.235,Z 388.291,A -85,B 0,C 180,E1 -9118.404,E2 -9118.404} C_VEL
LIN {X 0,Y 443.248,Z 383.956,A -85,B 0,C 180,E1 -9119.441,E2 -9119.441} C_VEL
LIN {X 0,Y 441.185,Z 374.05,A -85,B 0,C 180,E1 -9122.015,E2 -9122.015} C_VEL
LIN {X 0,Y 439.41,Z 365.753,A -85,B 0,C 180,E1 -9124.284,E2 -9124.284} C_VEL
LIN {X 0,Y 439.349,Z 365.757,A -85,B 0,C 180,E1 -9127.435,E2 -9127.435} C_VEL
LIN {X 0,Y 439.402,Z 365.752,A -85,B 0,C 180,E1 -9129.849,E2 -9129.849} C_VEL
LIN {X 0,Y 439.387,Z 365.753,A -85,B 0,C 180,E1 -9132.627,E2 -9132.627} C_VEL
LIN {X 0,Y 439.407,Z 365.751,A -85,B 0,C 180,E1 -9135.271,E2 -9135.271} C_VEL
LIN {X 0,Y 439.391,Z 365.752,A -85,B 0,C 180,E1 -9138.743,E2 -9138.743} C_VEL
LIN {X 0,Y 439.387,Z 365.753,A -85,B 0,C 180,E1 -9141.606,E2 -9141.606} C_VEL
LIN {X 0,Y 439.402,Z 365.752,A -85,B 0,C 180,E1 -9144.844,E2 -9144.844} C_VEL
LIN {X 0,Y 439.374,Z 365.756,A -85,B 0,C 180,E1 -9148.14,E2 -9148.14} C_VEL
LIN {X 0,Y 439.433,Z 365.747,A -85,B 0,C 180,E1 -9151.598,E2 -9151.598} C_VEL
LIN {X 0,Y 439.406,Z 365.75,A -85,B 0,C 180,E1 -9154.415,E2 -9154.415} C_VEL
LIN {X 0,Y 439.366,Z 365.757,A -85,B 0,C 180,E1 -9157.425,E2 -9157.425} C_VEL
LIN {X 0,Y 439.443,Z 365.745,A -85,B 0,C 180,E1 -9160.663,E2 -9160.663} C_VEL
LIN {X 0,Y 439.464,Z 365.743,A -85,B 0,C 180,E1 -9164.225,E2 -9164.225} C_VEL
LIN {X 0,Y 439.485,Z 365.742,A -85,B 0,C 180,E1 -9168.001,E2 -9168.001} C_VEL
LIN {X 0,Y 439.549,Z 365.736,A -85,B 0,C 180,E1 -9171.726,E2 -9171.726} C_VEL
LIN {X 0,Y 439.622,Z 365.722,A -85,B 0,C 180,E1 -9174.496,E2 -9174.496} C_VEL
LIN {X 0,Y 439.637,Z 365.723,A -85,B 0,C 180,E1 -9178.168,E2 -9178.168} C_VEL
LIN {X 0,Y 439.766,Z 365.708,A -85,B 0,C 180,E1 -9180,E2 -9180} C_VEL
LIN {X 0,Y 439.642,Z 365.72,A -85,B 0,C 180,E1 -9182.749,E2 -9182.749} C_VEL
LIN {X 0,Y 439.62,Z 365.723,A -85,B 0,C 180,E1 -9186.425,E2 -9186.425} C_VEL
LIN {X 0,Y 439.502,Z 365.739,A -85,B 0,C 180,E1 -9189.202,E2 -9189.202} C_VEL
LIN {X 0,Y 439.505,Z 365.738,A -85,B 0,C 180,E1 -9192.727,E2 -9192.727} C_VEL
LIN {X 0,Y 439.449,Z 365.743,A -85,B 0,C 180,E1 -9196.349,E2 -9196.349} C_VEL
LIN {X 0,Y 439.404,Z 365.751,A -85,B 0,C 180,E1 -9199.626,E2 -9199.626} C_VEL
LIN {X 0,Y 439.367,Z 365.756,A -85,B 0,C 180,E1 -9202.575,E2 -9202.575} C_VEL
LIN {X 0,Y 439.407,Z 365.75,A -85,B 0,C 180,E1 -9205.585,E2 -9205.585} C_VEL
LIN {X 0,Y 439.418,Z 365.751,A -85,B 0,C 180,E1 -9208.674,E2 -9208.674} C_VEL
LIN {X 0,Y 439.371,Z 365.755,A -85,B 0,C 180,E1 -9212.031,E2 -9212.031} C_VEL
LIN {X 0,Y 439.397,Z 365.753,A -85,B 0,C 180,E1 -9215.341,E2 -9215.341} C_VEL
LIN {X 0,Y 439.385,Z 365.755,A -85,B 0,C 180,E1 -9218.595,E2 -9218.595} C_VEL
LIN {X 0,Y 439.389,Z 365.753,A -85,B 0,C 180,E1 -9221.257,E2 -9221.257} C_VEL
LIN {X 0,Y 439.404,Z 365.752,A -85,B 0,C 180,E1 -9224.729,E2 -9224.729} C_VEL
LIN {X 0,Y 439.399,Z 365.749,A -85,B 0,C 180,E1 -9227.796,E2 -9227.796} C_VEL
LIN {X 0,Y 439.438,Z 365.747,A -85,B 0,C 180,E1 -9230.229,E2 -9230.229} C_VEL
LIN {X 0,Y 439.375,Z 365.755,A -85,B 0,C 180,E1 -9233.713,E2 -9233.713} C_VEL
LIN {X 0,Y 439.374,Z 365.755,A -85,B 0,C 180,E1 -9237.054,E2 -9237.054} C_VEL
LIN {X 0,Y 439.385,Z 365.755,A -85,B 0,C 180,E1 -9240.274,E2 -9240.274} C_VEL
LIN {X 0,Y 439.432,Z 365.747,A -85,B 0,C 180,E1 -9243.397,E2 -9243.397} C_VEL
LIN {X 0,Y 439.389,Z 365.754,A -85,B 0,C 180,E1 -9246.43,E2 -9246.43} C_VEL
LIN {X 0,Y 439.391,Z 365.751,A -85,B 0,C 180,E1 -9249.397,E2 -9249.397} C_VEL
LIN {X 0,Y 439.435,Z 365.749,A -85,B 0,C 180,E1 -9252.31,E2 -9252.31} C_VEL
LIN {X 0,Y 439.455,Z 365.745,A -85,B 0,C 180,E1 -9255.174,E2 -9255.174} C_VEL
LIN {X 0,Y 439.487,Z 365.741,A -85,B 0,C 180,E1 -9258.002,E2 -9258.002} C_VEL
LIN {X 0,Y 439.551,Z 365.732,A -85,B 0,C 180,E1 -9261.726,E2 -9261.726} C_VEL
LIN {X 0,Y 439.621,Z 365.724,A -85,B 0,C 180,E1 -9264.496,E2 -9264.496} C_VEL
LIN {X 0,Y 439.638,Z 365.723,A -85,B 0,C 180,E1 -9268.168,E2 -9268.168} C_VEL
LIN {X 0,Y 439.768,Z 365.707,A -85,B 0,C 180,E1 -9270,E2 -9270} C_VEL
LIN {X 0,Y 439.625,Z 365.722,A -85,B 0,C 180,E1 -9270.989,E2 -9270.989} C_VEL
LIN {X 0,Y 438.907,Z 365.815,A -85,B 0,C 180,E1 -9271.753,E2 -9271.753} C_VEL
LIN {X 0,Y 435.928,Z 366.181,A -85,B 0,C 180,E1 -9272.992,E2 -9272.992} C_VEL
LIN {X 0,Y 433.476,Z 366.491,A -85,B 0,C 180,E1 -9273.992,E2 -9273.992} C_VEL
LIN {X 0,Y 432.502,Z 366.61,A -85,B 0,C 180,E1 -9274.767,E2 -9274.767} C_VEL
LIN {X 0,Y 432.465,Z 366.614,A -85,B 0,C 180,E1 -9275.029,E2 -9275.029} C_VEL
LIN {X 0,Y 432.563,Z 366.604,A -85,B 0,C 180,E1 -9277.654,E2 -9277.654} C_VEL
LIN {X 0,Y 432.396,Z 366.623,A -85,B 0,C 180,E1 -9281.247,E2 -9281.247} C_VEL
LIN {X 0,Y 432.377,Z 366.626,A -85,B 0,C 180,E1 -9284.112,E2 -9284.112} C_VEL
LIN {X 0,Y 432.4,Z 366.623,A -85,B 0,C 180,E1 -9287.012,E2 -9287.012} C_VEL
LIN {X 0,Y 432.342,Z 366.632,A -85,B 0,C 180,E1 -9289.961,E2 -9289.961} C_VEL
LIN {X 0,Y 432.321,Z 366.632,A -85,B 0,C 180,E1 -9292.964,E2 -9292.964} C_VEL
LIN {X 0,Y 432.364,Z 366.627,A -85,B 0,C 180,E1 -9296.033,E2 -9296.033} C_VEL
LIN {X 0,Y 432.346,Z 366.632,A -85,B 0,C 180,E1 -9299.187,E2 -9299.187} C_VEL
LIN {X 0,Y 432.326,Z 366.632,A -85,B 0,C 180,E1 -9302.443,E2 -9302.443} C_VEL
LIN {X 0,Y 432.347,Z 366.631,A -85,B 0,C 180,E1 -9305.632,E2 -9305.632} C_VEL
LIN {X 0,Y 432.353,Z 366.63,A -85,B 0,C 180,E1 -9309.343,E2 -9309.343} C_VEL
LIN {X 0,Y 432.338,Z 366.633,A -85,B 0,C 180,E1 -9311.797,E2 -9311.797} C_VEL
LIN {X 0,Y 432.342,Z 366.63,A -85,B 0,C 180,E1 -9314.347,E2 -9314.347} C_VEL
LIN {X 0,Y 432.323,Z 366.635,A -85,B 0,C 180,E1 -9317.016,E2 -9317.016} C_VEL
LIN {X 0,Y 432.34,Z 366.631,A -85,B 0,C 180,E1 -9319.82,E2 -9319.82} C_VEL
LIN {X 0,Y 432.319,Z 366.634,A -85,B 0,C 180,E1 -9323.023,E2 -9323.023} C_VEL
LIN {X 0,Y 432.363,Z 366.626,A -85,B 0,C 180,E1 -9325.996,E2 -9325.996} C_VEL
LIN {X 0,Y 432.457,Z 366.644,A -85,B 0,C 180,E1 -9329.323,E2 -9329.323} C_VEL
LIN {X 0,Y 432.394,Z 371.489,A -85,B 0,C 180,E1 -9331.877,E2 -9331.877} C_VEL
LIN {X 0,Y 432.169,Z 377.481,A -85,B 0,C 180,E1 -9334.987,E2 -9334.987} C_VEL
LIN {X 0,Y 432.018,Z 383.432,A -85,B 0,C 180,E1 -9338.027,E2 -9338.027} C_VEL
LIN {X 0,Y 431.894,Z 389.384,A -85,B 0,C 180,E1 -9341.007,E2 -9341.007} C_VEL
LIN {X 0,Y 431.819,Z 395.261,A -85,B 0,C 180,E1 -9343.938,E2 -9343.938} C_VEL
LIN {X 0,Y 431.64,Z 403.149,A -85,B 0,C 180,E1 -9347.78,E2 -9347.78} C_VEL
LIN {X 0,Y 431.5,Z 407.843,A -85,B 0,C 180,E1 -9350.035,E2 -9350.035} C_VEL
LIN {X 0,Y 433.093,Z 418.667,A -85,B 0,C 180,E1 -9350.602,E2 -9350.602} C_VEL
LIN {X 0,Y 433.026,Z 428.143,A -85,B 0,C 180,E1 -9351.248,E2 -9351.248} C_VEL
LIN {X 0,Y 432.731,Z 436.439,A -85,B 0,C 180,E1 -9351.983,E2 -9351.983} C_VEL
LIN {X 0,Y 432.373,Z 444.87,A -85,B 0,C 180,E1 -9352.94,E2 -9352.94} C_VEL
LIN {X 0,Y 432.302,Z 451.637,A -85,B 0,C 180,E1 -9353.934,E2 -9353.934} C_VEL
LIN {X 0,Y 432.051,Z 457.819,A -85,B 0,C 180,E1 -9355.101,E2 -9355.101} C_VEL
LIN {X 0,Y 431.866,Z 462.451,A -85,B 0,C 180,E1 -9356.268,E2 -9356.268} C_VEL
LIN {X 0,Y 431.554,Z 466.34,A -85,B 0,C 180,E1 -9357.667,E2 -9357.667} C_VEL
LIN {X 0,Y 431.435,Z 468.581,A -85,B 0,C 180,E1 -9359.067,E2 -9359.067} C_VEL
LIN {X 0,Y 431.447,Z 469.218,A -85,B 0,C 180,E1 -9360,E2 -9360} C_VEL
LIN {X 0,Y 431.483,Z 469.183,A -85,B 0,C 180,E1 -9360.933,E2 -9360.933} C_VEL
LIN {X 0,Y 431.555,Z 468.478,A -85,B 0,C 180,E1 -9361.866,E2 -9361.866} C_VEL
LIN {X 0,Y 431.692,Z 467.096,A -85,B 0,C 180,E1 -9362.799,E2 -9362.799} C_VEL
LIN {X 0,Y 431.95,Z 465.006,A -85,B 0,C 180,E1 -9363.732,E2 -9363.732} C_VEL
LIN {X 0,Y 432.18,Z 462.17,A -85,B 0,C 180,E1 -9364.664,E2 -9364.664} C_VEL
LIN {X 0,Y 432.542,Z 457.416,A -85,B 0,C 180,E1 -9365.828,E2 -9365.828} C_VEL
LIN {X 0,Y 432.824,Z 451.128,A -85,B 0,C 180,E1 -9366.995,E2 -9366.995} C_VEL
LIN {X 0,Y 433.299,Z 444.159,A -85,B 0,C 180,E1 -9367.985,E2 -9367.985} C_VEL
LIN {X 0,Y 433.801,Z 435.233,A -85,B 0,C 180,E1 -9368.971,E2 -9368.971} C_VEL
LIN {X 0,Y 434.226,Z 425.514,A -85,B 0,C 180,E1 -9369.785,E2 -9369.785} C_VEL
LIN {X 0,Y 433.986,Z 420.417,A -85,B 0,C 180,E1 -9370.143,E2 -9370.143} C_VEL
LIN {X 0,Y 431.947,Z 410.627,A -85,B 0,C 180,E1 -9370.784,E2 -9370.784} C_VEL
LIN {X 0,Y 432.119,Z 406.064,A -85,B 0,C 180,E1 -9373.162,E2 -9373.162} C_VEL
LIN {X 0,Y 432.378,Z 399.887,A -85,B 0,C 180,E1 -9376.462,E2 -9376.462} C_VEL
LIN {X 0,Y 432.655,Z 393.57,A -85,B 0,C 180,E1 -9379.945,E2 -9379.945} C_VEL
LIN {X 0,Y 432.963,Z 388.356,A -85,B 0,C 180,E1 -9382.928,E2 -9382.928} C_VEL
LIN {X 0,Y 433.337,Z 383.249,A -85,B 0,C 180,E1 -9385.97,E2 -9385.97} C_VEL
LIN {X 0,Y 433.805,Z 378.28,A -85,B 0,C 180,E1 -9389.08,E2 -9389.08} C_VEL
LIN {X 0,Y 433.819,Z 375.187,A -85,B 0,C 180,E1 -9391.226,E2 -9391.226} C_VEL
LIN {X 0,Y 433.46,Z 372.281,A -85,B 0,C 180,E1 -9393.454,E2 -9393.454} C_VEL
LIN {X 0,Y 432.976,Z 369.715,A -85,B 0,C 180,E1 -9395.757,E2 -9395.757} C_VEL
LIN {X 0,Y 432.461,Z 367.129,A -85,B 0,C 180,E1 -9398.734,E2 -9398.734} C_VEL
LIN {X 0,Y 432.431,Z 366.622,A -85,B 0,C 180,E1 -9399.753,E2 -9399.753} C_VEL
LIN {X 0,Y 432.368,Z 366.629,A -85,B 0,C 180,E1 -9403.055,E2 -9403.055} C_VEL
LIN {X 0,Y 432.344,Z 366.632,A -85,B 0,C 180,E1 -9405.663,E2 -9405.663} C_VEL
LIN {X 0,Y 432.366,Z 366.759,A -85,B 0,C 180,E1 -9408.206,E2 -9408.206} C_VEL
LIN {X 0,Y 432.978,Z 369.252,A -85,B 0,C 180,E1 -9410.725,E2 -9410.725} C_VEL
LIN {X 0,Y 433.81,Z 372.806,A -85,B 0,C 180,E1 -9413.171,E2 -9413.171} C_VEL
LIN {X 0,Y 435.002,Z 377.354,A -85,B 0,C 180,E1 -9415.565,E2 -9415.565} C_VEL
LIN {X 0,Y 436.205,Z 382.769,A -85,B 0,C 180,E1 -9417.88,E2 -9417.88} C_VEL
LIN {X 0,Y 437.425,Z 389.157,A -85,B 0,C 180,E1 -9420.182,E2 -9420.182} C_VEL
LIN {X 0,Y 437.284,Z 392.349,A -85,B 0,C 180,E1 -9421.173,E2 -9421.173} C_VEL
LIN {X 0,Y 435.607,Z 403.277,A -85,B 0,C 180,E1 -9424.175,E2 -9424.175} C_VEL
LIN {X 0,Y 434.338,Z 415.453,A -85,B 0,C 180,E1 -9427.267,E2 -9427.267} C_VEL
LIN {X 0,Y 433.261,Z 429.538,A -85,B 0,C 180,E1 -9430.615,E2 -9430.615} C_VEL
LIN {X 0,Y 432.491,Z 443.259,A -85,B 0,C 180,E1 -9433.715,E2 -9433.715} C_VEL
LIN {X 0,Y 433.944,Z 455.682,A -85,B 0,C 180,E1 -9434.124,E2 -9434.124} C_VEL
LIN {X 0,Y 434.716,Z 467.666,A -85,B 0,C 180,E1 -9434.649,E2 -9434.649} C_VEL
LIN {X 0,Y 434.195,Z 480.269,A -85,B 0,C 180,E1 -9435.35,E2 -9435.35} C_VEL
LIN {X 0,Y 433.612,Z 491.454,A -85,B 0,C 180,E1 -9436.168,E2 -9436.168} C_VEL
LIN {X 0,Y 433.106,Z 501.747,A -85,B 0,C 180,E1 -9437.107,E2 -9437.107} C_VEL
LIN {X 0,Y 432.529,Z 510.212,A -85,B 0,C 180,E1 -9438.043,E2 -9438.043} C_VEL
LIN {X 0,Y 432.156,Z 519.026,A -85,B 0,C 180,E1 -9439.221,E2 -9439.221} C_VEL
LIN {X 0,Y 431.768,Z 527.556,A -85,B 0,C 180,E1 -9440.632,E2 -9440.632} C_VEL
LIN {X 0,Y 431.572,Z 534.427,A -85,B 0,C 180,E1 -9442.043,E2 -9442.043} C_VEL
LIN {X 0,Y 431.465,Z 540.136,A -85,B 0,C 180,E1 -9443.521,E2 -9443.521} C_VEL
LIN {X 0,Y 431.411,Z 544.131,A -85,B 0,C 180,E1 -9444.859,E2 -9444.859} C_VEL
LIN {X 0,Y 431.486,Z 547.267,A -85,B 0,C 180,E1 -9446.264,E2 -9446.264} C_VEL
LIN {X 0,Y 431.501,Z 548.764,A -85,B 0,C 180,E1 -9447.199,E2 -9447.199} C_VEL
LIN {X 0,Y 431.426,Z 549.825,A -85,B 0,C 180,E1 -9448.133,E2 -9448.133} C_VEL
LIN {X 0,Y 431.348,Z 550.477,A -85,B 0,C 180,E1 -9449.066,E2 -9449.066} C_VEL
LIN {X 0,Y 431.339,Z 550.691,A -85,B 0,C 180,E1 -9450,E2 -9450} C_VEL
LIN {X 0,Y 431.424,Z 549.843,A -85,B 0,C 180,E1 -9451.867,E2 -9451.867} C_VEL
LIN {X 0,Y 431.546,Z 548.801,A -85,B 0,C 180,E1 -9452.8,E2 -9452.8} C_VEL
LIN {X 0,Y 431.469,Z 547.256,A -85,B 0,C 180,E1 -9453.736,E2 -9453.736} C_VEL
LIN {X 0,Y 431.404,Z 544.097,A -85,B 0,C 180,E1 -9455.14,E2 -9455.14} C_VEL
LIN {X 0,Y 431.482,Z 539.82,A -85,B 0,C 180,E1 -9456.547,E2 -9456.547} C_VEL
LIN {X 0,Y 431.563,Z 534.285,A -85,B 0,C 180,E1 -9457.956,E2 -9457.956} C_VEL
LIN {X 0,Y 431.77,Z 527.311,A -85,B 0,C 180,E1 -9459.368,E2 -9459.368} C_VEL
LIN {X 0,Y 432.154,Z 518.492,A -85,B 0,C 180,E1 -9460.779,E2 -9460.779} C_VEL
LIN {X 0,Y 432.511,Z 509.395,A -85,B 0,C 180,E1 -9461.957,E2 -9461.957} C_VEL
LIN {X 0,Y 432.996,Z 501.401,A -85,B 0,C 180,E1 -9462.81,E2 -9462.81} C_VEL
LIN {X 0,Y 433.458,Z 491.599,A -85,B 0,C 180,E1 -9463.681,E2 -9463.681} C_VEL
LIN {X 0,Y 433.931,Z 481.293,A -85,B 0,C 180,E1 -9464.419,E2 -9464.419} C_VEL
LIN {X 0,Y 434.394,Z 469.657,A -85,B 0,C 180,E1 -9465.062,E2 -9465.062} C_VEL
LIN {X 0,Y 434.237,Z 463.54,A -85,B 0,C 180,E1 -9465.338,E2 -9465.338} C_VEL
LIN {X 0,Y 433.02,Z 449.926,A -85,B 0,C 180,E1 -9465.82,E2 -9465.82} C_VEL
LIN {X 0,Y 432.403,Z 444.243,A -85,B 0,C 180,E1 -9465.979,E2 -9465.979} C_VEL
LIN {X 0,Y 433.04,Z 430.993,A -85,B 0,C 180,E1 -9468.941,E2 -9468.941} C_VEL
LIN {X 0,Y 433.905,Z 418.048,A -85,B 0,C 180,E1 -9471.872,E2 -9471.872} C_VEL
LIN {X 0,Y 435.106,Z 402.39,A -85,B 0,C 180,E1 -9475.472,E2 -9475.472} C_VEL
LIN {X 0,Y 436.345,Z 389.025,A -85,B 0,C 180,E1 -9478.631,E2 -9478.631} C_VEL
LIN {X 0,Y 436.299,Z 385.257,A -85,B 0,C 180,E1 -9479.559,E2 -9479.559} C_VEL
LIN {X 0,Y 434.366,Z 375.999,A -85,B 0,C 180,E1 -9481.998,E2 -9481.998} C_VEL
LIN {X 0,Y 432.38,Z 366.628,A -85,B 0,C 180,E1 -9484.586,E2 -9484.586} C_VEL
LIN {X 0,Y 432.338,Z 366.631,A -85,B 0,C 180,E1 -9488.15,E2 -9488.15} C_VEL
LIN {X 0,Y 432.336,Z 366.634,A -85,B 0,C 180,E1 -9491.602,E2 -9491.602} C_VEL
LIN {X 0,Y 432.342,Z 366.631,A -85,B 0,C 180,E1 -9494.346,E2 -9494.346} C_VEL
LIN {X 0,Y 432.326,Z 366.632,A -85,B 0,C 180,E1 -9497.015,E2 -9497.015} C_VEL
LIN {X 0,Y 432.343,Z 366.63,A -85,B 0,C 180,E1 -9499.819,E2 -9499.819} C_VEL
LIN {X 0,Y 432.317,Z 366.633,A -85,B 0,C 180,E1 -9503.023,E2 -9503.023} C_VEL
LIN {X 0,Y 432.361,Z 366.629,A -85,B 0,C 180,E1 -9505.996,E2 -9505.996} C_VEL
LIN {X 0,Y 432.348,Z 366.629,A -85,B 0,C 180,E1 -9509.489,E2 -9509.489} C_VEL
LIN {X 0,Y 432.393,Z 366.623,A -85,B 0,C 180,E1 -9512.928,E2 -9512.928} C_VEL
LIN {X 0,Y 432.372,Z 366.627,A -85,B 0,C 180,E1 -9516.023,E2 -9516.023} C_VEL
LIN {X 0,Y 432.351,Z 366.629,A -85,B 0,C 180,E1 -9519.046,E2 -9519.046} C_VEL
LIN {X 0,Y 432.38,Z 366.627,A -85,B 0,C 180,E1 -9522.011,E2 -9522.011} C_VEL
LIN {X 0,Y 432.398,Z 366.623,A -85,B 0,C 180,E1 -9524.927,E2 -9524.927} C_VEL
LIN {X 0,Y 432.46,Z 366.616,A -85,B 0,C 180,E1 -9527.803,E2 -9527.803} C_VEL
LIN {X 0,Y 432.493,Z 366.613,A -85,B 0,C 180,E1 -9531.59,E2 -9531.59} C_VEL
LIN {X 0,Y 432.599,Z 366.597,A -85,B 0,C 180,E1 -9534.406,E2 -9534.406} C_VEL
LIN {X 0,Y 432.607,Z 366.599,A -85,B 0,C 180,E1 -9538.138,E2 -9538.138} C_VEL
LIN {X 0,Y 432.735,Z 366.583,A -85,B 0,C 180,E1 -9540,E2 -9540} C_VEL
LIN {X 0,Y 432.594,Z 366.598,A -85,B 0,C 180,E1 -9542.794,E2 -9542.794} C_VEL
LIN {X 0,Y 432.574,Z 366.6,A -85,B 0,C 180,E1 -9546.53,E2 -9546.53} C_VEL
LIN {X 0,Y 432.446,Z 366.618,A -85,B 0,C 180,E1 -9549.353,E2 -9549.353} C_VEL
LIN {X 0,Y 432.446,Z 366.617,A -85,B 0,C 180,E1 -9552.812,E2 -9552.812} C_VEL
LIN {X 0,Y 432.414,Z 366.62,A -85,B 0,C 180,E1 -9556.479,E2 -9556.479} C_VEL
LIN {X 0,Y 432.34,Z 366.631,A -85,B 0,C 180,E1 -9559.96,E2 -9559.96} C_VEL
LIN {X 0,Y 432.321,Z 366.634,A -85,B 0,C 180,E1 -9562.964,E2 -9562.964} C_VEL
LIN {X 0,Y 432.365,Z 366.625,A -85,B 0,C 180,E1 -9566.032,E2 -9566.032} C_VEL
LIN {X 0,Y 432.344,Z 366.631,A -85,B 0,C 180,E1 -9569.188,E2 -9569.188} C_VEL
LIN {X 0,Y 432.324,Z 366.634,A -85,B 0,C 180,E1 -9572.443,E2 -9572.443} C_VEL
LIN {X 0,Y 432.346,Z 366.629,A -85,B 0,C 180,E1 -9575.632,E2 -9575.632} C_VEL
LIN {X 0,Y 432.348,Z 366.633,A -85,B 0,C 180,E1 -9578.716,E2 -9578.716} C_VEL
LIN {X 0,Y 432.334,Z 366.631,A -85,B 0,C 180,E1 -9581.797,E2 -9581.797} C_VEL
LIN {X 0,Y 432.335,Z 366.632,A -85,B 0,C 180,E1 -9584.347,E2 -9584.347} C_VEL
LIN {X 0,Y 432.326,Z 366.634,A -85,B 0,C 180,E1 -9587.015,E2 -9587.015} C_VEL
LIN {X 0,Y 432.343,Z 366.629,A -85,B 0,C 180,E1 -9589.82,E2 -9589.82} C_VEL
LIN {X 0,Y 432.308,Z 366.635,A -85,B 0,C 180,E1 -9593.022,E2 -9593.022} C_VEL
LIN {X 0,Y 432.361,Z 366.629,A -85,B 0,C 180,E1 -9595.997,E2 -9595.997} C_VEL
LIN {X 0,Y 432.349,Z 366.627,A -85,B 0,C 180,E1 -9599.49,E2 -9599.49} C_VEL
LIN {X 0,Y 432.394,Z 366.624,A -85,B 0,C 180,E1 -9602.929,E2 -9602.929} C_VEL
LIN {X 0,Y 432.373,Z 366.627,A -85,B 0,C 180,E1 -9606.024,E2 -9606.024} C_VEL
LIN {X 0,Y 432.353,Z 366.628,A -85,B 0,C 180,E1 -9609.046,E2 -9609.046} C_VEL
LIN {X 0,Y 432.382,Z 366.627,A -85,B 0,C 180,E1 -9612.011,E2 -9612.011} C_VEL
LIN {X 0,Y 432.405,Z 366.623,A -85,B 0,C 180,E1 -9614.927,E2 -9614.927} C_VEL
LIN {X 0,Y 432.462,Z 366.616,A -85,B 0,C 180,E1 -9617.804,E2 -9617.804} C_VEL
LIN {X 0,Y 432.495,Z 366.61,A -85,B 0,C 180,E1 -9621.591,E2 -9621.591} C_VEL
LIN {X 0,Y 432.597,Z 366.599,A -85,B 0,C 180,E1 -9624.406,E2 -9624.406} C_VEL
LIN {X 0,Y 432.608,Z 366.598,A -85,B 0,C 180,E1 -9628.138,E2 -9628.138} C_VEL
LIN {X 0,Y 432.737,Z 366.583,A -85,B 0,C 180,E1 -9630,E2 -9630} C_VEL
LIN {X 0,Y 432.595,Z 366.596,A -85,B 0,C 180,E1 -9632.794,E2 -9632.794} C_VEL
LIN {X 0,Y 432.465,Z 366.614,A -85,B 0,C 180,E1 -9635.029,E2 -9635.029} C_VEL
LIN {X 0,Y 431.905,Z 366.687,A -85,B 0,C 180,E1 -9635.807,E2 -9635.807} C_VEL
LIN {X 0,Y 429.06,Z 367.039,A -85,B 0,C 180,E1 -9637.071,E2 -9637.071} C_VEL
LIN {X 0,Y 426.578,Z 367.35,A -85,B 0,C 180,E1 -9638.092,E2 -9638.092} C_VEL
LIN {X 0,Y 425.497,Z 367.483,A -85,B 0,C 180,E1 -9638.882,E2 -9638.882} C_VEL
LIN {X 0,Y 425.406,Z 367.493,A -85,B 0,C 180,E1 -9639.149,E2 -9639.149} C_VEL
LIN {X 0,Y 425.397,Z 367.494,A -85,B 0,C 180,E1 -9642.904,E2 -9642.904} C_VEL
LIN {X 0,Y 425.365,Z 367.499,A -85,B 0,C 180,E1 -9646.605,E2 -9646.605} C_VEL
LIN {X 0,Y 425.332,Z 367.504,A -85,B 0,C 180,E1 -9649.636,E2 -9649.636} C_VEL
LIN {X 0,Y 425.308,Z 367.507,A -85,B 0,C 180,E1 -9653.365,E2 -9653.365} C_VEL
LIN {X 0,Y 425.351,Z 367.501,A -85,B 0,C 180,E1 -9656.844,E2 -9656.844} C_VEL
LIN {X 0,Y 425.294,Z 367.509,A -85,B 0,C 180,E1 -9659.72,E2 -9659.72} C_VEL
LIN {X 0,Y 425.285,Z 367.509,A -85,B 0,C 180,E1 -9663.048,E2 -9663.048} C_VEL
LIN {X 0,Y 425.285,Z 367.508,A -85,B 0,C 180,E1 -9665.929,E2 -9665.929} C_VEL
LIN {X 0,Y 425.301,Z 367.51,A -85,B 0,C 180,E1 -9669.044,E2 -9669.044} C_VEL
LIN {X 0,Y 425.281,Z 367.511,A -85,B 0,C 180,E1 -9672.653,E2 -9672.653} C_VEL
LIN {X 0,Y 425.264,Z 367.51,A -85,B 0,C 180,E1 -9676.044,E2 -9676.044} C_VEL
LIN {X 0,Y 425.278,Z 367.51,A -85,B 0,C 180,E1 -9678.622,E2 -9678.622} C_VEL
LIN {X 0,Y 425.316,Z 367.507,A -85,B 0,C 180,E1 -9681.103,E2 -9681.103} C_VEL
LIN {X 0,Y 425.304,Z 367.507,A -85,B 0,C 180,E1 -9684.664,E2 -9684.664} C_VEL
LIN {X 0,Y 425.336,Z 367.503,A -85,B 0,C 180,E1 -9688.079,E2 -9688.079} C_VEL
LIN {X 0,Y 425.43,Z 367.589,A -85,B 0,C 180,E1 -9689.297,E2 -9689.297} C_VEL
LIN {X 0,Y 425.414,Z 371.474,A -85,B 0,C 180,E1 -9691.374,E2 -9691.374} C_VEL
LIN {X 0,Y 425.155,Z 377.526,A -85,B 0,C 180,E1 -9694.546,E2 -9694.546} C_VEL
LIN {X 0,Y 424.968,Z 383.906,A -85,B 0,C 180,E1 -9697.837,E2 -9697.837} C_VEL
LIN {X 0,Y 424.86,Z 389.481,A -85,B 0,C 180,E1 -9700.68,E2 -9700.68} C_VEL
LIN {X 0,Y 424.74,Z 395.464,A -85,B 0,C 180,E1 -9703.68,E2 -9703.68} C_VEL
LIN {X 0,Y 424.568,Z 403.419,A -85,B 0,C 180,E1 -9707.594,E2 -9707.594} C_VEL
LIN {X 0,Y 424.418,Z 408.103,A -85,B 0,C 180,E1 -9709.867,E2 -9709.867} C_VEL
LIN {X 0,Y 426.114,Z 419.755,A -85,B 0,C 180,E1 -9710.507,E2 -9710.507} C_VEL
LIN {X 0,Y 425.938,Z 429.776,A -85,B 0,C 180,E1 -9711.221,E2 -9711.221} C_VEL
LIN {X 0,Y 425.573,Z 439.05,A -85,B 0,C 180,E1 -9712.097,E2 -9712.097} C_VEL
LIN {X 0,Y 425.304,Z 446.588,A -85,B 0,C 180,E1 -9713.012,E2 -9713.012} C_VEL
LIN {X 0,Y 425.216,Z 453.418,A -85,B 0,C 180,E1 -9714.071,E2 -9714.071} C_VEL
LIN {X 0,Y 424.977,Z 459.332,A -85,B 0,C 180,E1 -9715.257,E2 -9715.257} C_VEL
LIN {X 0,Y 424.806,Z 462.973,A -85,B 0,C 180,E1 -9716.206,E2 -9716.206} C_VEL
LIN {X 0,Y 424.498,Z 466.927,A -85,B 0,C 180,E1 -9717.628,E2 -9717.628} C_VEL
LIN {X 0,Y 424.371,Z 469.228,A -85,B 0,C 180,E1 -9719.051,E2 -9719.051} C_VEL
LIN {X 0,Y 424.381,Z 469.908,A -85,B 0,C 180,E1 -9720,E2 -9720} C_VEL
LIN {X 0,Y 424.423,Z 469.921,A -85,B 0,C 180,E1 -9720.949,E2 -9720.949} C_VEL
LIN {X 0,Y 424.504,Z 469.268,A -85,B 0,C 180,E1 -9721.897,E2 -9721.897} C_VEL
LIN {X 0,Y 424.651,Z 467.939,A -85,B 0,C 180,E1 -9722.846,E2 -9722.846} C_VEL
LIN {X 0,Y 424.923,Z 465.899,A -85,B 0,C 180,E1 -9723.793,E2 -9723.793} C_VEL
LIN {X 0,Y 425.168,Z 463.116,A -85,B 0,C 180,E1 -9724.741,E2 -9724.741} C_VEL
LIN {X 0,Y 425.552,Z 458.448,A -85,B 0,C 180,E1 -9725.925,E2 -9725.925} C_VEL
LIN {X 0,Y 425.876,Z 452.263,A -85,B 0,C 180,E1 -9727.11,E2 -9727.11} C_VEL
LIN {X 0,Y 426.394,Z 445.148,A -85,B 0,C 180,E1 -9728.152,E2 -9728.152} C_VEL
LIN {X 0,Y 426.919,Z 436.753,A -85,B 0,C 180,E1 -9729.116,E2 -9729.116} C_VEL
LIN {X 0,Y 427.394,Z 427.444,A -85,B 0,C 180,E1 -9729.943,E2 -9729.943} C_VEL
LIN {X 0,Y 427.336,Z 422.613,A -85,B 0,C 180,E1 -9730.303,E2 -9730.303} C_VEL
LIN {X 0,Y 425.442,Z 413.274,A -85,B 0,C 180,E1 -9730.951,E2 -9730.951} C_VEL
LIN {X 0,Y 424.93,Z 411.115,A -85,B 0,C 180,E1 -9731.085,E2 -9731.085} C_VEL
LIN {X 0,Y 425.113,Z 406.796,A -85,B 0,C 180,E1 -9733.382,E2 -9733.382} C_VEL
LIN {X 0,Y 425.396,Z 400.841,A -85,B 0,C 180,E1 -9736.619,E2 -9736.619} C_VEL
LIN {X 0,Y 425.675,Z 395.26,A -85,B 0,C 180,E1 -9739.765,E2 -9739.765} C_VEL
LIN {X 0,Y 426.06,Z 389.177,A -85,B 0,C 180,E1 -9743.321,E2 -9743.321} C_VEL
LIN {X 0,Y 426.498,Z 384.113,A -85,B 0,C 180,E1 -9746.418,E2 -9746.418} C_VEL
LIN {X 0,Y 426.945,Z 379.295,A -85,B 0,C 180,E1 -9749.593,E2 -9749.593} C_VEL
LIN {X 0,Y 426.905,Z 376.277,A -85,B 0,C 180,E1 -9751.79,E2 -9751.79} C_VEL
LIN {X 0,Y 426.462,Z 373.048,A -85,B 0,C 180,E1 -9754.513,E2 -9754.513} C_VEL
LIN {X 0,Y 425.9,Z 370.197,A -85,B 0,C 180,E1 -9757.63,E2 -9757.63} C_VEL
LIN {X 0,Y 425.56,Z 368.592,A -85,B 0,C 180,E1 -9760.096,E2 -9760.096} C_VEL
LIN {X 0,Y 425.344,Z 367.761,A -85,B 0,C 180,E1 -9762.645,E2 -9762.645} C_VEL
LIN {X 0,Y 425.362,Z 367.903,A -85,B 0,C 180,E1 -9765.273,E2 -9765.273} C_VEL
LIN {X 0,Y 425.742,Z 369.187,A -85,B 0,C 180,E1 -9767.974,E2 -9767.974} C_VEL
LIN {X 0,Y 426.405,Z 371.926,A -85,B 0,C 180,E1 -9770.774,E2 -9770.774} C_VEL
LIN {X 0,Y 426.927,Z 374.279,A -85,B 0,C 180,E1 -9772.476,E2 -9772.476} C_VEL
LIN {X 0,Y 428.167,Z 379.035,A -85,B 0,C 180,E1 -9775.156,E2 -9775.156} C_VEL
LIN {X 0,Y 429.243,Z 383.682,A -85,B 0,C 180,E1 -9777.295,E2 -9777.295} C_VEL
LIN {X 0,Y 430.532,Z 390.508,A -85,B 0,C 180,E1 -9779.903,E2 -9779.903} C_VEL
LIN {X 0,Y 430.604,Z 392.893,A -85,B 0,C 180,E1 -9780.683,E2 -9780.683} C_VEL
LIN {X 0,Y 429.163,Z 401.719,A -85,B 0,C 180,E1 -9783.234,E2 -9783.234} C_VEL
LIN {X 0,Y 427.715,Z 413.144,A -85,B 0,C 180,E1 -9786.261,E2 -9786.261} C_VEL
LIN {X 0,Y 426.589,Z 426.187,A -85,B 0,C 180,E1 -9789.507,E2 -9789.507} C_VEL
LIN {X 0,Y 425.603,Z 441.483,A -85,B 0,C 180,E1 -9793.089,E2 -9793.089} C_VEL
LIN {X 0,Y 425.526,Z 442.911,A -85,B 0,C 180,E1 -9793.415,E2 -9793.415} C_VEL
LIN {X 0,Y 427.039,Z 455.374,A -85,B 0,C 180,E1 -9793.845,E2 -9793.845} C_VEL
LIN {X 0,Y 427.831,Z 468.722,A -85,B 0,C 180,E1 -9794.456,E2 -9794.456} C_VEL
LIN {X 0,Y 427.32,Z 479.919,A -85,B 0,C 180,E1 -9795.109,E2 -9795.109} C_VEL
LIN {X 0,Y 426.67,Z 491.04,A -85,B 0,C 180,E1 -9795.939,E2 -9795.939} C_VEL
LIN {X 0,Y 426.142,Z 500.679,A -85,B 0,C 180,E1 -9796.832,E2 -9796.832} C_VEL
LIN {X 0,Y 425.552,Z 509.691,A -85,B 0,C 180,E1 -9797.844,E2 -9797.844} C_VEL
LIN {X 0,Y 425.139,Z 518.468,A -85,B 0,C 180,E1 -9799.041,E2 -9799.041} C_VEL
LIN {X 0,Y 424.722,Z 526.973,A -85,B 0,C 180,E1 -9800.475,E2 -9800.475} C_VEL
LIN {X 0,Y 424.515,Z 533.823,A -85,B 0,C 180,E1 -9801.91,E2 -9801.91} C_VEL
LIN {X 0,Y 424.385,Z 539.88,A -85,B 0,C 180,E1 -9803.529,E2 -9803.529} C_VEL
LIN {X 0,Y 424.349,Z 543.501,A -85,B 0,C 180,E1 -9804.773,E2 -9804.773} C_VEL
LIN {X 0,Y 424.399,Z 546.622,A -85,B 0,C 180,E1 -9806.202,E2 -9806.202} C_VEL
LIN {X 0,Y 424.424,Z 548.107,A -85,B 0,C 180,E1 -9807.152,E2 -9807.152} C_VEL
LIN {X 0,Y 424.373,Z 549.164,A -85,B 0,C 180,E1 -9808.102,E2 -9808.102} C_VEL
LIN {X 0,Y 424.289,Z 549.809,A -85,B 0,C 180,E1 -9809.051,E2 -9809.051} C_VEL
LIN {X 0,Y 424.277,Z 550.002,A -85,B 0,C 180,E1 -9810,E2 -9810} C_VEL
LIN {X 0,Y 424.372,Z 549.137,A -85,B 0,C 180,E1 -9811.898,E2 -9811.898} C_VEL
LIN {X 0,Y 424.477,Z 548.067,A -85,B 0,C 180,E1 -9812.847,E2 -9812.847} C_VEL
LIN {X 0,Y 424.307,Z 545.573,A -85,B 0,C 180,E1 -9814.274,E2 -9814.274} C_VEL
LIN {X 0,Y 424.374,Z 542.021,A -85,B 0,C 180,E1 -9815.702,E2 -9815.702} C_VEL
LIN {X 0,Y 424.429,Z 537.281,A -85,B 0,C 180,E1 -9817.134,E2 -9817.134} C_VEL
LIN {X 0,Y 424.581,Z 531.218,A -85,B 0,C 180,E1 -9818.567,E2 -9818.567} C_VEL
LIN {X 0,Y 424.803,Z 523.603,A -85,B 0,C 180,E1 -9820.004,E2 -9820.004} C_VEL
LIN {X 0,Y 425.215,Z 515.768,A -85,B 0,C 180,E1 -9821.198,E2 -9821.198} C_VEL
LIN {X 0,Y 425.733,Z 506.124,A -85,B 0,C 180,E1 -9822.392,E2 -9822.392} C_VEL
LIN {X 0,Y 426.13,Z 496.66,A -85,B 0,C 180,E1 -9823.35,E2 -9823.35} C_VEL
LIN {X 0,Y 426.761,Z 484.899,A -85,B 0,C 180,E1 -9824.301,E2 -9824.301} C_VEL
LIN {X 0,Y 427.308,Z 472.283,A -85,B 0,C 180,E1 -9825.074,E2 -9825.074} C_VEL
LIN {X 0,Y 427.455,Z 466.185,A -85,B 0,C 180,E1 -9825.374,E2 -9825.374} C_VEL
LIN {X 0,Y 426.415,Z 454.201,A -85,B 0,C 180,E1 -9825.857,E2 -9825.857} C_VEL
LIN {X 0,Y 425.354,Z 443.983,A -85,B 0,C 180,E1 -9826.159,E2 -9826.159} C_VEL
LIN {X 0,Y 426.075,Z 430.39,A -85,B 0,C 180,E1 -9829.262,E2 -9829.262} C_VEL
LIN {X 0,Y 427.079,Z 416.17,A -85,B 0,C 180,E1 -9832.56,E2 -9832.56} C_VEL
LIN {X 0,Y 428.321,Z 401.417,A -85,B 0,C 180,E1 -9836.049,E2 -9836.049} C_VEL
LIN {X 0,Y 429.45,Z 389.718,A -85,B 0,C 180,E1 -9838.866,E2 -9838.866} C_VEL
LIN {X 0,Y 429.238,Z 386.026,A -85,B 0,C 180,E1 -9839.798,E2 -9839.798} C_VEL
LIN {X 0,Y 427.243,Z 376.766,A -85,B 0,C 180,E1 -9842.307,E2 -9842.307} C_VEL
LIN {X 0,Y 425.32,Z 367.508,A -85,B 0,C 180,E1 -9844.931,E2 -9844.931} C_VEL
LIN {X 0,Y 425.307,Z 367.507,A -85,B 0,C 180,E1 -9848.898,E2 -9848.898} C_VEL
LIN {X 0,Y 425.293,Z 367.511,A -85,B 0,C 180,E1 -9851.958,E2 -9851.958} C_VEL
LIN {X 0,Y 425.292,Z 367.508,A -85,B 0,C 180,E1 -9855.282,E2 -9855.282} C_VEL
LIN {X 0,Y 425.299,Z 367.508,A -85,B 0,C 180,E1 -9858.624,E2 -9858.624} C_VEL
LIN {X 0,Y 425.317,Z 367.503,A -85,B 0,C 180,E1 -9861.103,E2 -9861.103} C_VEL
LIN {X 0,Y 425.301,Z 367.509,A -85,B 0,C 180,E1 -9864.664,E2 -9864.664} C_VEL
LIN {X 0,Y 425.266,Z 367.513,A -85,B 0,C 180,E1 -9868.073,E2 -9868.073} C_VEL
LIN {X 0,Y 425.332,Z 367.502,A -85,B 0,C 180,E1 -9871.368,E2 -9871.368} C_VEL
LIN {X 0,Y 425.296,Z 367.508,A -85,B 0,C 180,E1 -9874.555,E2 -9874.555} C_VEL
LIN {X 0,Y 425.289,Z 367.51,A -85,B 0,C 180,E1 -9877.661,E2 -9877.661} C_VEL
LIN {X 0,Y 425.363,Z 367.498,A -85,B 0,C 180,E1 -9880.704,E2 -9880.704} C_VEL
LIN {X 0,Y 425.39,Z 367.5,A -85,B 0,C 180,E1 -9883.688,E2 -9883.688} C_VEL
LIN {X 0,Y 425.413,Z 367.494,A -85,B 0,C 180,E1 -9887.598,E2 -9887.598} C_VEL
LIN {X 0,Y 425.444,Z 367.49,A -85,B 0,C 180,E1 -9891.45,E2 -9891.45} C_VEL
LIN {X 0,Y 425.555,Z 367.474,A -85,B 0,C 180,E1 -9894.313,E2 -9894.313} C_VEL
LIN {X 0,Y 425.577,Z 367.474,A -85,B 0,C 180,E1 -9898.107,E2 -9898.107} C_VEL
LIN {X 0,Y 425.705,Z 367.459,A -85,B 0,C 180,E1 -9900,E2 -9900} C_VEL
LIN {X 0,Y 425.547,Z 367.476,A -85,B 0,C 180,E1 -9902.84,E2 -9902.84} C_VEL
LIN {X 0,Y 425.532,Z 367.478,A -85,B 0,C 180,E1 -9906.644,E2 -9906.644} C_VEL
LIN {X 0,Y 425.405,Z 367.495,A -85,B 0,C 180,E1 -9909.509,E2 -9909.509} C_VEL
LIN {X 0,Y 425.405,Z 367.494,A -85,B 0,C 180,E1 -9912.91,E2 -9912.91} C_VEL
LIN {X 0,Y 425.363,Z 367.499,A -85,B 0,C 180,E1 -9916.605,E2 -9916.605} C_VEL
LIN {X 0,Y 425.33,Z 367.505,A -85,B 0,C 180,E1 -9919.636,E2 -9919.636} C_VEL
LIN {X 0,Y 425.309,Z 367.51,A -85,B 0,C 180,E1 -9923.365,E2 -9923.365} C_VEL
LIN {X 0,Y 425.348,Z 367.503,A -85,B 0,C 180,E1 -9926.844,E2 -9926.844} C_VEL
LIN {X 0,Y 425.292,Z 367.509,A -85,B 0,C 180,E1 -9929.72,E2 -9929.72} C_VEL
LIN {X 0,Y 425.283,Z 367.511,A -85,B 0,C 180,E1 -9933.048,E2 -9933.048} C_VEL
LIN {X 0,Y 425.286,Z 367.508,A -85,B 0,C 180,E1 -9935.929,E2 -9935.929} C_VEL
LIN {X 0,Y 425.299,Z 367.509,A -85,B 0,C 180,E1 -9939.044,E2 -9939.044} C_VEL
LIN {X 0,Y 425.276,Z 367.512,A -85,B 0,C 180,E1 -9942.653,E2 -9942.653} C_VEL
LIN {X 0,Y 425.27,Z 367.511,A -85,B 0,C 180,E1 -9946.045,E2 -9946.045} C_VEL
LIN {X 0,Y 425.286,Z 367.508,A -85,B 0,C 180,E1 -9949.479,E2 -9949.479} C_VEL
LIN {X 0,Y 425.28,Z 367.512,A -85,B 0,C 180,E1 -9952.489,E2 -9952.489} C_VEL
LIN {X 0,Y 425.309,Z 367.507,A -85,B 0,C 180,E1 -9955.818,E2 -9955.818} C_VEL
LIN {X 0,Y 425.292,Z 367.506,A -85,B 0,C 180,E1 -9959.239,E2 -9959.239} C_VEL
LIN {X 0,Y 425.352,Z 367.503,A -85,B 0,C 180,E1 -9962.443,E2 -9962.443} C_VEL
LIN {X 0,Y 425.353,Z 367.501,A -85,B 0,C 180,E1 -9965.602,E2 -9965.602} C_VEL
LIN {X 0,Y 425.296,Z 367.51,A -85,B 0,C 180,E1 -9968.682,E2 -9968.682} C_VEL
LIN {X 0,Y 425.336,Z 367.502,A -85,B 0,C 180,E1 -9971.703,E2 -9971.703} C_VEL
LIN {X 0,Y 425.359,Z 367.501,A -85,B 0,C 180,E1 -9974.671,E2 -9974.671} C_VEL
LIN {X 0,Y 425.415,Z 367.494,A -85,B 0,C 180,E1 -9977.598,E2 -9977.598} C_VEL
LIN {X 0,Y 425.445,Z 367.487,A -85,B 0,C 180,E1 -9981.45,E2 -9981.45} C_VEL
LIN {X 0,Y 425.554,Z 367.477,A -85,B 0,C 180,E1 -9984.313,E2 -9984.313} C_VEL
LIN {X 0,Y 425.577,Z 367.474,A -85,B 0,C 180,E1 -9988.107,E2 -9988.107} C_VEL
LIN {X 0,Y 425.707,Z 367.459,A -85,B 0,C 180,E1 -9990,E2 -9990} C_VEL
LIN {X 0,Y 425.549,Z 367.474,A -85,B 0,C 180,E1 -9992.84,E2 -9992.84} C_VEL
LIN {X 0,Y 425.526,Z 367.48,A -85,B 0,C 180,E1 -9996.639,E2 -9996.639} C_VEL
LIN {X 0,Y 425.406,Z 367.493,A -85,B 0,C 180,E1 -9999.149,E2 -9999.149} C_VEL
LIN {X 0,Y 424.734,Z 367.58,A -85,B 0,C 180,E1 -9999.939,E2 -9999.939} C_VEL
LIN {X 0,Y 421.886,Z 367.933,A -85,B 0,C 180,E1 -10001.223,E2 -10001.223} C_VEL
LIN {X 0,Y 419.47,Z 368.234,A -85,B 0,C 180,E1 -10002.259,E2 -10002.259} C_VEL
LIN {X 0,Y 418.419,Z 368.363,A -85,B 0,C 180,E1 -10003.06,E2 -10003.06} C_VEL
LIN {X 0,Y 418.326,Z 368.376,A -85,B 0,C 180,E1 -10003.331,E2 -10003.331} C_VEL
LIN {X 0,Y 418.316,Z 368.377,A -85,B 0,C 180,E1 -10006.736,E2 -10006.736} C_VEL
LIN {X 0,Y 418.274,Z 368.384,A -85,B 0,C 180,E1 -10009.791,E2 -10009.791} C_VEL
LIN {X 0,Y 418.241,Z 368.386,A -85,B 0,C 180,E1 -10012.736,E2 -10012.736} C_VEL
LIN {X 0,Y 418.272,Z 368.383,A -85,B 0,C 180,E1 -10015.904,E2 -10015.904} C_VEL
LIN {X 0,Y 418.268,Z 368.386,A -85,B 0,C 180,E1 -10019.162,E2 -10019.162} C_VEL
LIN {X 0,Y 418.261,Z 368.385,A -85,B 0,C 180,E1 -10022.844,E2 -10022.844} C_VEL
LIN {X 0,Y 418.248,Z 368.384,A -85,B 0,C 180,E1 -10026.238,E2 -10026.238} C_VEL
LIN {X 0,Y 418.255,Z 368.386,A -85,B 0,C 180,E1 -10029.682,E2 -10029.682} C_VEL
LIN {X 0,Y 418.235,Z 368.387,A -85,B 0,C 180,E1 -10032.322,E2 -10032.322} C_VEL
LIN {X 0,Y 418.24,Z 368.388,A -85,B 0,C 180,E1 -10035.109,E2 -10035.109} C_VEL
LIN {X 0,Y 418.243,Z 368.386,A -85,B 0,C 180,E1 -10037.767,E2 -10037.767} C_VEL
LIN {X 0,Y 418.26,Z 368.385,A -85,B 0,C 180,E1 -10040.619,E2 -10040.619} C_VEL
LIN {X 0,Y 418.249,Z 368.385,A -85,B 0,C 180,E1 -10043.976,E2 -10043.976} C_VEL
LIN {X 0,Y 418.269,Z 368.387,A -85,B 0,C 180,E1 -10047.154,E2 -10047.154} C_VEL
LIN {X 0,Y 418.39,Z 368.481,A -85,B 0,C 180,E1 -10049.247,E2 -10049.247} C_VEL
LIN {X 0,Y 418.386,Z 372.471,A -85,B 0,C 180,E1 -10051.403,E2 -10051.403} C_VEL
LIN {X 0,Y 418.111,Z 378.538,A -85,B 0,C 180,E1 -10054.619,E2 -10054.619} C_VEL
LIN {X 0,Y 417.923,Z 384.337,A -85,B 0,C 180,E1 -10057.655,E2 -10057.655} C_VEL
LIN {X 0,Y 417.815,Z 389.661,A -85,B 0,C 180,E1 -10060.385,E2 -10060.385} C_VEL
LIN {X 0,Y 417.627,Z 397.579,A -85,B 0,C 180,E1 -10064.38,E2 -10064.38} C_VEL
LIN {X 0,Y 417.485,Z 403.91,A -85,B 0,C 180,E1 -10067.524,E2 -10067.524} C_VEL
LIN {X 0,Y 417.369,Z 408.451,A -85,B 0,C 180,E1 -10069.724,E2 -10069.724} C_VEL
LIN {X 0,Y 418.834,Z 418.808,A -85,B 0,C 180,E1 -10070.279,E2 -10070.279} C_VEL
LIN {X 0,Y 419.161,Z 423.566,A -85,B 0,C 180,E1 -10070.591,E2 -10070.591} C_VEL
LIN {X 0,Y 418.79,Z 432.753,A -85,B 0,C 180,E1 -10071.313,E2 -10071.313} C_VEL
LIN {X 0,Y 418.449,Z 442.064,A -85,B 0,C 180,E1 -10072.278,E2 -10072.278} C_VEL
LIN {X 0,Y 418.241,Z 449.324,A -85,B 0,C 180,E1 -10073.245,E2 -10073.245} C_VEL
LIN {X 0,Y 418.042,Z 456.364,A -85,B 0,C 180,E1 -10074.453,E2 -10074.453} C_VEL
LIN {X 0,Y 417.903,Z 461.712,A -85,B 0,C 180,E1 -10075.66,E2 -10075.66} C_VEL
LIN {X 0,Y 417.561,Z 466.325,A -85,B 0,C 180,E1 -10077.106,E2 -10077.106} C_VEL
LIN {X 0,Y 417.382,Z 468.449,A -85,B 0,C 180,E1 -10078.07,E2 -10078.07} C_VEL
LIN {X 0,Y 417.31,Z 469.864,A -85,B 0,C 180,E1 -10079.035,E2 -10079.035} C_VEL
LIN {X 0,Y 417.316,Z 470.6,A -85,B 0,C 180,E1 -10080,E2 -10080} C_VEL
LIN {X 0,Y 417.364,Z 470.664,A -85,B 0,C 180,E1 -10080.965,E2 -10080.965} C_VEL
LIN {X 0,Y 417.453,Z 470.062,A -85,B 0,C 180,E1 -10081.93,E2 -10081.93} C_VEL
LIN {X 0,Y 417.611,Z 468.783,A -85,B 0,C 180,E1 -10082.894,E2 -10082.894} C_VEL
LIN {X 0,Y 418.168,Z 465.505,A -85,B 0,C 180,E1 -10084.337,E2 -10084.337} C_VEL
LIN {X 0,Y 418.28,Z 462.404,A -85,B 0,C 180,E1 -10085.302,E2 -10085.302} C_VEL
LIN {X 0,Y 418.692,Z 457.292,A -85,B 0,C 180,E1 -10086.506,E2 -10086.506} C_VEL
LIN {X 0,Y 419.203,Z 450.547,A -85,B 0,C 180,E1 -10087.708,E2 -10087.708} C_VEL
LIN {X 0,Y 419.685,Z 443.635,A -85,B 0,C 180,E1 -10088.668,E2 -10088.668} C_VEL
LIN {X 0,Y 420.247,Z 434.828,A -85,B 0,C 180,E1 -10089.627,E2 -10089.627} C_VEL
LIN {X 0,Y 420.641,Z 424.794,A -85,B 0,C 180,E1 -10090.469,E2 -10090.469} C_VEL
LIN {X 0,Y 418.97,Z 415.97,A -85,B 0,C 180,E1 -10091.122,E2 -10091.122} C_VEL
LIN {X 0,Y 417.948,Z 411.582,A -85,B 0,C 180,E1 -10091.426,E2 -10091.426} C_VEL
LIN {X 0,Y 418.132,Z 407.544,A -85,B 0,C 180,E1 -10093.61,E2 -10093.61} C_VEL
LIN {X 0,Y 418.413,Z 401.841,A -85,B 0,C 180,E1 -10096.779,E2 -10096.779} C_VEL
LIN {X 0,Y 418.742,Z 396.314,A -85,B 0,C 180,E1 -10099.967,E2 -10099.967} C_VEL
LIN {X 0,Y 419.048,Z 391.689,A -85,B 0,C 180,E1 -10102.716,E2 -10102.716} C_VEL
LIN {X 0,Y 419.452,Z 386.695,A -85,B 0,C 180,E1 -10105.826,E2 -10105.826} C_VEL
LIN {X 0,Y 420.021,Z 381.866,A -85,B 0,C 180,E1 -10109.028,E2 -10109.028} C_VEL
LIN {X 0,Y 420.107,Z 378.625,A -85,B 0,C 180,E1 -10111.44,E2 -10111.44} C_VEL
LIN {X 0,Y 419.815,Z 376.138,A -85,B 0,C 180,E1 -10113.535,E2 -10113.535} C_VEL
LIN {X 0,Y 419.284,Z 373.365,A -85,B 0,C 180,E1 -10116.431,E2 -10116.431} C_VEL
LIN {X 0,Y 418.923,Z 371.157,A -85,B 0,C 180,E1 -10119.606,E2 -10119.606} C_VEL
LIN {X 0,Y 418.712,Z 370.242,A -85,B 0,C 180,E1 -10122.393,E2 -10122.393} C_VEL
LIN {X 0,Y 418.728,Z 370.418,A -85,B 0,C 180,E1 -10125.175,E2 -10125.175} C_VEL
LIN {X 0,Y 419.12,Z 371.738,A -85,B 0,C 180,E1 -10127.875,E2 -10127.875} C_VEL
LIN {X 0,Y 419.706,Z 374.166,A -85,B 0,C 180,E1 -10130.482,E2 -10130.482} C_VEL
LIN {X 0,Y 420.63,Z 378.201,A -85,B 0,C 180,E1 -10133.321,E2 -10133.321} C_VEL
LIN {X 0,Y 421.67,Z 382.136,A -85,B 0,C 180,E1 -10135.481,E2 -10135.481} C_VEL
LIN {X 0,Y 422.85,Z 387.656,A -85,B 0,C 180,E1 -10137.957,E2 -10137.957} C_VEL
LIN {X 0,Y 423.853,Z 393.487,A -85,B 0,C 180,E1 -10140.169,E2 -10140.169} C_VEL
LIN {X 0,Y 423.079,Z 398.866,A -85,B 0,C 180,E1 -10141.831,E2 -10141.831} C_VEL
LIN {X 0,Y 421.18,Z 411.407,A -85,B 0,C 180,E1 -10145.344,E2 -10145.344} C_VEL
LIN {X 0,Y 419.813,Z 424.136,A -85,B 0,C 180,E1 -10148.647,E2 -10148.647} C_VEL
LIN {X 0,Y 418.787,Z 438.593,A -85,B 0,C 180,E1 -10152.165,E2 -10152.165} C_VEL
LIN {X 0,Y 418.542,Z 442.603,A -85,B 0,C 180,E1 -10153.101,E2 -10153.101} C_VEL
LIN {X 0,Y 420.231,Z 455.736,A -85,B 0,C 180,E1 -10153.576,E2 -10153.576} C_VEL
LIN {X 0,Y 420.997,Z 468.691,A -85,B 0,C 180,E1 -10154.198,E2 -10154.198} C_VEL
LIN {X 0,Y 420.35,Z 481.431,A -85,B 0,C 180,E1 -10154.98,E2 -10154.98} C_VEL
LIN {X 0,Y 419.675,Z 492.129,A -85,B 0,C 180,E1 -10155.823,E2 -10155.823} C_VEL
LIN {X 0,Y 419.07,Z 502.604,A -85,B 0,C 180,E1 -10156.859,E2 -10156.859} C_VEL
LIN {X 0,Y 418.367,Z 512.913,A -85,B 0,C 180,E1 -10158.124,E2 -10158.124} C_VEL
LIN {X 0,Y 417.914,Z 520.996,A -85,B 0,C 180,E1 -10159.34,E2 -10159.34} C_VEL
LIN {X 0,Y 417.569,Z 528.87,A -85,B 0,C 180,E1 -10160.799,E2 -10160.799} C_VEL
LIN {X 0,Y 417.371,Z 535.18,A -85,B 0,C 180,E1 -10162.258,E2 -10162.258} C_VEL
LIN {X 0,Y 417.287,Z 539.708,A -85,B 0,C 180,E1 -10163.56,E2 -10163.56} C_VEL
LIN {X 0,Y 417.225,Z 544.007,A -85,B 0,C 180,E1 -10165.168,E2 -10165.168} C_VEL
LIN {X 0,Y 417.301,Z 545.98,A -85,B 0,C 180,E1 -10166.137,E2 -10166.137} C_VEL
LIN {X 0,Y 417.349,Z 547.455,A -85,B 0,C 180,E1 -10167.104,E2 -10167.104} C_VEL
LIN {X 0,Y 417.32,Z 548.505,A -85,B 0,C 180,E1 -10168.07,E2 -10168.07} C_VEL
LIN {X 0,Y 417.232,Z 549.138,A -85,B 0,C 180,E1 -10169.035,E2 -10169.035} C_VEL
LIN {X 0,Y 417.217,Z 549.31,A -85,B 0,C 180,E1 -10170,E2 -10170} C_VEL
LIN {X 0,Y 417.23,Z 549.065,A -85,B 0,C 180,E1 -10170.965,E2 -10170.965} C_VEL
LIN {X 0,Y 417.321,Z 548.421,A -85,B 0,C 180,E1 -10171.93,E2 -10171.93} C_VEL
LIN {X 0,Y 417.41,Z 547.315,A -85,B 0,C 180,E1 -10172.895,E2 -10172.895} C_VEL
LIN {X 0,Y 417.241,Z 544.783,A -85,B 0,C 180,E1 -10174.347,E2 -10174.347} C_VEL
LIN {X 0,Y 417.259,Z 540.368,A -85,B 0,C 180,E1 -10176.074,E2 -10176.074} C_VEL
LIN {X 0,Y 417.38,Z 534.526,A -85,B 0,C 180,E1 -10177.742,E2 -10177.742} C_VEL
LIN {X 0,Y 417.569,Z 527.883,A -85,B 0,C 180,E1 -10179.2,E2 -10179.2} C_VEL
LIN {X 0,Y 417.897,Z 519.57,A -85,B 0,C 180,E1 -10180.661,E2 -10180.661} C_VEL
LIN {X 0,Y 418.325,Z 510.961,A -85,B 0,C 180,E1 -10181.876,E2 -10181.876} C_VEL
LIN {X 0,Y 418.864,Z 501.68,A -85,B 0,C 180,E1 -10182.946,E2 -10182.946} C_VEL
LIN {X 0,Y 419.429,Z 491.08,A -85,B 0,C 180,E1 -10183.938,E2 -10183.938} C_VEL
LIN {X 0,Y 419.98,Z 479.619,A -85,B 0,C 180,E1 -10184.785,E2 -10184.785} C_VEL
LIN {X 0,Y 420.493,Z 467.751,A -85,B 0,C 180,E1 -10185.449,E2 -10185.449} C_VEL
LIN {X 0,Y 419.516,Z 456.155,A -85,B 0,C 180,E1 -10185.953,E2 -10185.953} C_VEL
LIN {X 0,Y 418.342,Z 443.716,A -85,B 0,C 180,E1 -10186.343,E2 -10186.343} C_VEL
LIN {X 0,Y 419.098,Z 429.82,A -85,B 0,C 180,E1 -10189.596,E2 -10189.596} C_VEL
LIN {X 0,Y 420.056,Z 417.007,A -85,B 0,C 180,E1 -10192.632,E2 -10192.632} C_VEL
LIN {X 0,Y 421.373,Z 402.061,A -85,B 0,C 180,E1 -10196.231,E2 -10196.231} C_VEL
LIN {X 0,Y 422.528,Z 390.388,A -85,B 0,C 180,E1 -10199.112,E2 -10199.112} C_VEL
LIN {X 0,Y 422.177,Z 386.826,A -85,B 0,C 180,E1 -10200.043,E2 -10200.043} C_VEL
LIN {X 0,Y 419.808,Z 375.514,A -85,B 0,C 180,E1 -10203.17,E2 -10203.17} C_VEL
LIN {X 0,Y 418.28,Z 368.384,A -85,B 0,C 180,E1 -10205.28,E2 -10205.28} C_VEL
LIN {X 0,Y 418.254,Z 368.386,A -85,B 0,C 180,E1 -10208.442,E2 -10208.442} C_VEL
LIN {X 0,Y 418.223,Z 368.388,A -85,B 0,C 180,E1 -10210.948,E2 -10210.948} C_VEL
LIN {X 0,Y 418.218,Z 368.391,A -85,B 0,C 180,E1 -10213.73,E2 -10213.73} C_VEL
LIN {X 0,Y 418.217,Z 368.392,A -85,B 0,C 180,E1 -10216.449,E2 -10216.449} C_VEL
LIN {X 0,Y 418.261,Z 368.382,A -85,B 0,C 180,E1 -10219.124,E2 -10219.124} C_VEL
LIN {X 0,Y 418.236,Z 368.389,A -85,B 0,C 180,E1 -10222.165,E2 -10222.165} C_VEL
LIN {X 0,Y 418.267,Z 368.384,A -85,B 0,C 180,E1 -10225.42,E2 -10225.42} C_VEL
LIN {X 0,Y 418.212,Z 368.391,A -85,B 0,C 180,E1 -10228.604,E2 -10228.604} C_VEL
LIN {X 0,Y 418.293,Z 368.384,A -85,B 0,C 180,E1 -10231.937,E2 -10231.937} C_VEL
LIN {X 0,Y 418.29,Z 368.381,A -85,B 0,C 180,E1 -10235.163,E2 -10235.163} C_VEL
LIN {X 0,Y 418.235,Z 368.389,A -85,B 0,C 180,E1 -10238.304,E2 -10238.304} C_VEL
LIN {X 0,Y 418.285,Z 368.381,A -85,B 0,C 180,E1 -10241.383,E2 -10241.383} C_VEL
LIN {X 0,Y 418.304,Z 368.378,A -85,B 0,C 180,E1 -10244.406,E2 -10244.406} C_VEL
LIN {X 0,Y 418.357,Z 368.374,A -85,B 0,C 180,E1 -10247.386,E2 -10247.386} C_VEL
LIN {X 0,Y 418.343,Z 368.374,A -85,B 0,C 180,E1 -10250.329,E2 -10250.329} C_VEL
LIN {X 0,Y 418.495,Z 368.355,A -85,B 0,C 180,E1 -10253.249,E2 -10253.249} C_VEL
LIN {X 0,Y 418.342,Z 368.375,A -85,B 0,C 180,E1 -10255.182,E2 -10255.182} C_VEL
LIN {X 0,Y 418.546,Z 368.35,A -85,B 0,C 180,E1 -10258.075,E2 -10258.075} C_VEL
LIN {X 0,Y 418.674,Z 368.334,A -85,B 0,C 180,E1 -10260,E2 -10260} C_VEL
LIN {X 0,Y 418.502,Z 368.354,A -85,B 0,C 180,E1 -10262.888,E2 -10262.888} C_VEL
LIN {X 0,Y 418.495,Z 368.355,A -85,B 0,C 180,E1 -10266.751,E2 -10266.751} C_VEL
LIN {X 0,Y 418.361,Z 368.373,A -85,B 0,C 180,E1 -10269.671,E2 -10269.671} C_VEL
LIN {X 0,Y 418.356,Z 368.373,A -85,B 0,C 180,E1 -10273.006,E2 -10273.006} C_VEL
LIN {X 0,Y 418.314,Z 368.378,A -85,B 0,C 180,E1 -10276.736,E2 -10276.736} C_VEL
LIN {X 0,Y 418.272,Z 368.384,A -85,B 0,C 180,E1 -10279.791,E2 -10279.791} C_VEL
LIN {X 0,Y 418.239,Z 368.388,A -85,B 0,C 180,E1 -10282.736,E2 -10282.736} C_VEL
LIN {X 0,Y 418.272,Z 368.381,A -85,B 0,C 180,E1 -10285.904,E2 -10285.904} C_VEL
LIN {X 0,Y 418.266,Z 368.385,A -85,B 0,C 180,E1 -10289.162,E2 -10289.162} C_VEL
LIN {X 0,Y 418.258,Z 368.386,A -85,B 0,C 180,E1 -10292.844,E2 -10292.844} C_VEL
LIN {X 0,Y 418.249,Z 368.385,A -85,B 0,C 180,E1 -10296.239,E2 -10296.239} C_VEL
LIN {X 0,Y 418.252,Z 368.384,A -85,B 0,C 180,E1 -10299.682,E2 -10299.682} C_VEL
LIN {X 0,Y 418.231,Z 368.39,A -85,B 0,C 180,E1 -10302.321,E2 -10302.321} C_VEL
LIN {X 0,Y 418.241,Z 368.389,A -85,B 0,C 180,E1 -10305.109,E2 -10305.109} C_VEL
LIN {X 0,Y 418.244,Z 368.384,A -85,B 0,C 180,E1 -10307.767,E2 -10307.767} C_VEL
LIN {X 0,Y 418.26,Z 368.387,A -85,B 0,C 180,E1 -10310.619,E2 -10310.619} C_VEL
LIN {X 0,Y 418.244,Z 368.387,A -85,B 0,C 180,E1 -10313.976,E2 -10313.976} C_VEL
LIN {X 0,Y 418.259,Z 368.384,A -85,B 0,C 180,E1 -10317.156,E2 -10317.156} C_VEL
LIN {X 0,Y 418.27,Z 368.383,A -85,B 0,C 180,E1 -10320.896,E2 -10320.896} C_VEL
LIN {X 0,Y 418.273,Z 368.385,A -85,B 0,C 180,E1 -10324.096,E2 -10324.096} C_VEL
LIN {X 0,Y 418.24,Z 368.386,A -85,B 0,C 180,E1 -10327.264,E2 -10327.264} C_VEL
LIN {X 0,Y 418.319,Z 368.381,A -85,B 0,C 180,E1 -10330.366,E2 -10330.366} C_VEL
LIN {X 0,Y 418.329,Z 368.375,A -85,B 0,C 180,E1 -10333.405,E2 -10333.405} C_VEL
LIN {X 0,Y 418.349,Z 368.373,A -85,B 0,C 180,E1 -10336.999,E2 -10336.999} C_VEL
LIN {X 0,Y 418.36,Z 368.375,A -85,B 0,C 180,E1 -10340.329,E2 -10340.329} C_VEL
LIN {X 0,Y 418.49,Z 368.354,A -85,B 0,C 180,E1 -10343.249,E2 -10343.249} C_VEL
LIN {X 0,Y 418.342,Z 368.374,A -85,B 0,C 180,E1 -10345.182,E2 -10345.182} C_VEL
LIN {X 0,Y 418.546,Z 368.35,A -85,B 0,C 180,E1 -10348.076,E2 -10348.076} C_VEL
LIN {X 0,Y 418.676,Z 368.334,A -85,B 0,C 180,E1 -10350,E2 -10350} C_VEL
LIN {X 0,Y 418.504,Z 368.352,A -85,B 0,C 180,E1 -10352.888,E2 -10352.888} C_VEL
LIN {X 0,Y 418.49,Z 368.356,A -85,B 0,C 180,E1 -10356.751,E2 -10356.751} C_VEL
LIN {X 0,Y 418.345,Z 368.375,A -85,B 0,C 180,E1 -10359.671,E2 -10359.671} C_VEL
LIN {X 0,Y 418.326,Z 368.376,A -85,B 0,C 180,E1 -10363.331,E2 -10363.331} C_VEL
LIN {X 0,Y 417.632,Z 368.466,A -85,B 0,C 180,E1 -10364.134,E2 -10364.134} C_VEL
LIN {X 0,Y 414.754,Z 368.823,A -85,B 0,C 180,E1 -10365.44,E2 -10365.44} C_VEL
LIN {X 0,Y 412.341,Z 369.121,A -85,B 0,C 180,E1 -10366.494,E2 -10366.494} C_VEL
LIN {X 0,Y 411.319,Z 369.251,A -85,B 0,C 180,E1 -10367.309,E2 -10367.309} C_VEL
LIN {X 0,Y 411.243,Z 369.257,A -85,B 0,C 180,E1 -10367.585,E2 -10367.585} C_VEL
LIN {X 0,Y 411.2,Z 369.264,A -85,B 0,C 180,E1 -10371.034,E2 -10371.034} C_VEL
LIN {X 0,Y 411.228,Z 369.259,A -85,B 0,C 180,E1 -10374.216,E2 -10374.216} C_VEL
LIN {X 0,Y 411.262,Z 369.258,A -85,B 0,C 180,E1 -10377.478,E2 -10377.478} C_VEL
LIN {X 0,Y 411.192,Z 369.265,A -85,B 0,C 180,E1 -10380.848,E2 -10380.848} C_VEL
LIN {X 0,Y 411.209,Z 369.261,A -85,B 0,C 180,E1 -10384.334,E2 -10384.334} C_VEL
LIN {X 0,Y 411.198,Z 369.264,A -85,B 0,C 180,E1 -10387.974,E2 -10387.974} C_VEL
LIN {X 0,Y 411.185,Z 369.265,A -85,B 0,C 180,E1 -10390.504,E2 -10390.504} C_VEL
LIN {X 0,Y 411.18,Z 369.267,A -85,B 0,C 180,E1 -10393.133,E2 -10393.133} C_VEL
LIN {X 0,Y 411.171,Z 369.266,A -85,B 0,C 180,E1 -10395.881,E2 -10395.881} C_VEL
LIN {X 0,Y 411.167,Z 369.269,A -85,B 0,C 180,E1 -10398.772,E2 -10398.772} C_VEL
LIN {X 0,Y 411.214,Z 369.262,A -85,B 0,C 180,E1 -10401.83,E2 -10401.83} C_VEL
LIN {X 0,Y 411.215,Z 369.264,A -85,B 0,C 180,E1 -10405.121,E2 -10405.121} C_VEL
LIN {X 0,Y 411.364,Z 369.338,A -85,B 0,C 180,E1 -10409.167,E2 -10409.167} C_VEL
LIN {X 0,Y 411.359,Z 373.459,A -85,B 0,C 180,E1 -10411.421,E2 -10411.421} C_VEL
LIN {X 0,Y 411.041,Z 380.119,A -85,B 0,C 180,E1 -10414.986,E2 -10414.986} C_VEL
LIN {X 0,Y 410.817,Z 386.672,A -85,B 0,C 180,E1 -10418.419,E2 -10418.419} C_VEL
LIN {X 0,Y 410.671,Z 392.706,A -85,B 0,C 180,E1 -10421.543,E2 -10421.543} C_VEL
LIN {X 0,Y 410.535,Z 398.711,A -85,B 0,C 180,E1 -10424.612,E2 -10424.612} C_VEL
LIN {X 0,Y 410.383,Z 405.771,A -85,B 0,C 180,E1 -10428.141,E2 -10428.141} C_VEL
LIN {X 0,Y 410.316,Z 408.733,A -85,B 0,C 180,E1 -10429.577,E2 -10429.577} C_VEL
LIN {X 0,Y 411.828,Z 419.639,A -85,B 0,C 180,E1 -10430.174,E2 -10430.174} C_VEL
LIN {X 0,Y 412.1,Z 425.162,A -85,B 0,C 180,E1 -10430.552,E2 -10430.552} C_VEL
LIN {X 0,Y 411.75,Z 434.059,A -85,B 0,C 180,E1 -10431.287,E2 -10431.287} C_VEL
LIN {X 0,Y 411.376,Z 443.12,A -85,B 0,C 180,E1 -10432.259,E2 -10432.259} C_VEL
LIN {X 0,Y 411.157,Z 451.133,A -85,B 0,C 180,E1 -10433.374,E2 -10433.374} C_VEL
LIN {X 0,Y 410.976,Z 457.916,A -85,B 0,C 180,E1 -10434.603,E2 -10434.603} C_VEL
LIN {X 0,Y 410.836,Z 462.146,A -85,B 0,C 180,E1 -10435.585,E2 -10435.585} C_VEL
LIN {X 0,Y 410.491,Z 466.849,A -85,B 0,C 180,E1 -10437.056,E2 -10437.056} C_VEL
LIN {X 0,Y 410.331,Z 469.03,A -85,B 0,C 180,E1 -10438.037,E2 -10438.037} C_VEL
LIN {X 0,Y 410.25,Z 470.503,A -85,B 0,C 180,E1 -10439.018,E2 -10439.018} C_VEL
LIN {X 0,Y 410.252,Z 471.292,A -85,B 0,C 180,E1 -10440,E2 -10440} C_VEL
LIN {X 0,Y 410.305,Z 471.409,A -85,B 0,C 180,E1 -10440.981,E2 -10440.981} C_VEL
LIN {X 0,Y 410.403,Z 470.861,A -85,B 0,C 180,E1 -10441.963,E2 -10441.963} C_VEL
LIN {X 0,Y 410.574,Z 469.645,A -85,B 0,C 180,E1 -10442.944,E2 -10442.944} C_VEL
LIN {X 0,Y 411.152,Z 466.477,A -85,B 0,C 180,E1 -10444.412,E2 -10444.412} C_VEL
LIN {X 0,Y 411.304,Z 463.459,A -85,B 0,C 180,E1 -10445.393,E2 -10445.393} C_VEL
LIN {X 0,Y 411.753,Z 458.461,A -85,B 0,C 180,E1 -10446.616,E2 -10446.616} C_VEL
LIN {X 0,Y 412.288,Z 451.858,A -85,B 0,C 180,E1 -10447.838,E2 -10447.838} C_VEL
LIN {X 0,Y 412.877,Z 443.931,A -85,B 0,C 180,E1 -10448.964,E2 -10448.964} C_VEL
LIN {X 0,Y 413.471,Z 435.347,A -85,B 0,C 180,E1 -10449.91,E2 -10449.91} C_VEL
LIN {X 0,Y 413.914,Z 426.993,A -85,B 0,C 180,E1 -10450.641,E2 -10450.641} C_VEL
LIN {X 0,Y 412.571,Z 418.838,A -85,B 0,C 180,E1 -10451.297,E2 -10451.297} C_VEL
LIN {X 0,Y 410.967,Z 412.069,A -85,B 0,C 180,E1 -10451.779,E2 -10451.779} C_VEL
LIN {X 0,Y 411.136,Z 408.333,A -85,B 0,C 180,E1 -10453.846,E2 -10453.846} C_VEL
LIN {X 0,Y 411.455,Z 402.842,A -85,B 0,C 180,E1 -10456.955,E2 -10456.955} C_VEL
LIN {X 0,Y 411.793,Z 397.38,A -85,B 0,C 180,E1 -10460.169,E2 -10460.169} C_VEL
LIN {X 0,Y 412.147,Z 392.633,A -85,B 0,C 180,E1 -10463.092,E2 -10463.092} C_VEL
LIN {X 0,Y 412.611,Z 387.665,A -85,B 0,C 180,E1 -10466.286,E2 -10466.286} C_VEL
LIN {X 0,Y 413.03,Z 384.483,A -85,B 0,C 180,E1 -10468.453,E2 -10468.453} C_VEL
LIN {X 0,Y 413.236,Z 381.488,A -85,B 0,C 180,E1 -10470.678,E2 -10470.678} C_VEL
LIN {X 0,Y 413.071,Z 378.762,A -85,B 0,C 180,E1 -10472.987,E2 -10472.987} C_VEL
LIN {X 0,Y 412.714,Z 376.412,A -85,B 0,C 180,E1 -10475.379,E2 -10475.379} C_VEL
LIN {X 0,Y 412.318,Z 374.208,A -85,B 0,C 180,E1 -10478.364,E2 -10478.364} C_VEL
LIN {X 0,Y 412.117,Z 373.202,A -85,B 0,C 180,E1 -10480.393,E2 -10480.393} C_VEL
LIN {X 0,Y 412.052,Z 372.68,A -85,B 0,C 180,E1 -10483.019,E2 -10483.019} C_VEL
LIN {X 0,Y 412.146,Z 373.209,A -85,B 0,C 180,E1 -10485.741,E2 -10485.741} C_VEL
LIN {X 0,Y 412.627,Z 374.858,A -85,B 0,C 180,E1 -10488.541,E2 -10488.541} C_VEL
LIN {X 0,Y 413.362,Z 377.957,A -85,B 0,C 180,E1 -10491.453,E2 -10491.453} C_VEL
LIN {X 0,Y 414.542,Z 382.661,A -85,B 0,C 180,E1 -10494.467,E2 -10494.467} C_VEL
LIN {X 0,Y 415.841,Z 388.353,A -85,B 0,C 180,E1 -10497.26,E2 -10497.26} C_VEL
LIN {X 0,Y 416.898,Z 394.189,A -85,B 0,C 180,E1 -10499.62,E2 -10499.62} C_VEL
LIN {X 0,Y 416.848,Z 397.41,A -85,B 0,C 180,E1 -10500.729,E2 -10500.729} C_VEL
LIN {X 0,Y 414.929,Z 407.956,A -85,B 0,C 180,E1 -10503.871,E2 -10503.871} C_VEL
LIN {X 0,Y 413.481,Z 419.283,A -85,B 0,C 180,E1 -10506.987,E2 -10506.987} C_VEL
LIN {X 0,Y 412.257,Z 432.281,A -85,B 0,C 180,E1 -10510.324,E2 -10510.324} C_VEL
LIN {X 0,Y 411.594,Z 442.401,A -85,B 0,C 180,E1 -10512.765,E2 -10512.765} C_VEL
LIN {X 0,Y 413.394,Z 455.482,A -85,B 0,C 180,E1 -10513.263,E2 -10513.263} C_VEL
LIN {X 0,Y 414.124,Z 467.667,A -85,B 0,C 180,E1 -10513.865,E2 -10513.865} C_VEL
LIN {X 0,Y 413.6,Z 479.625,A -85,B 0,C 180,E1 -10514.603,E2 -10514.603} C_VEL
LIN {X 0,Y 412.753,Z 491.9,A -85,B 0,C 180,E1 -10515.58,E2 -10515.58} C_VEL
LIN {X 0,Y 412.069,Z 502.933,A -85,B 0,C 180,E1 -10516.712,E2 -10516.712} C_VEL
LIN {X 0,Y 411.376,Z 512.498,A -85,B 0,C 180,E1 -10517.92,E2 -10517.92} C_VEL
LIN {X 0,Y 410.894,Z 520.524,A -85,B 0,C 180,E1 -10519.155,E2 -10519.155} C_VEL
LIN {X 0,Y 410.526,Z 528.338,A -85,B 0,C 180,E1 -10520.64,E2 -10520.64} C_VEL
LIN {X 0,Y 410.297,Z 534.622,A -85,B 0,C 180,E1 -10522.124,E2 -10522.124} C_VEL
LIN {X 0,Y 410.214,Z 539.458,A -85,B 0,C 180,E1 -10523.56,E2 -10523.56} C_VEL
LIN {X 0,Y 410.161,Z 543.395,A -85,B 0,C 180,E1 -10525.085,E2 -10525.085} C_VEL
LIN {X 0,Y 410.206,Z 545.341,A -85,B 0,C 180,E1 -10526.07,E2 -10526.07} C_VEL
LIN {X 0,Y 410.275,Z 546.806,A -85,B 0,C 180,E1 -10527.054,E2 -10527.054} C_VEL
LIN {X 0,Y 410.269,Z 547.849,A -85,B 0,C 180,E1 -10528.036,E2 -10528.036} C_VEL
LIN {X 0,Y 410.177,Z 548.46,A -85,B 0,C 180,E1 -10529.018,E2 -10529.018} C_VEL
LIN {X 0,Y 410.159,Z 548.609,A -85,B 0,C 180,E1 -10530,E2 -10530} C_VEL
LIN {X 0,Y 410.175,Z 548.351,A -85,B 0,C 180,E1 -10530.982,E2 -10530.982} C_VEL
LIN {X 0,Y 410.272,Z 547.69,A -85,B 0,C 180,E1 -10531.963,E2 -10531.963} C_VEL
LIN {X 0,Y 410.346,Z 546.547,A -85,B 0,C 180,E1 -10532.945,E2 -10532.945} C_VEL
LIN {X 0,Y 410.178,Z 543.973,A -85,B 0,C 180,E1 -10534.422,E2 -10534.422} C_VEL
LIN {X 0,Y 410.202,Z 540.321,A -85,B 0,C 180,E1 -10535.9,E2 -10535.9} C_VEL
LIN {X 0,Y 410.279,Z 535.472,A -85,B 0,C 180,E1 -10537.381,E2 -10537.381} C_VEL
LIN {X 0,Y 410.44,Z 529.278,A -85,B 0,C 180,E1 -10538.865,E2 -10538.865} C_VEL
LIN {X 0,Y 410.703,Z 521.448,A -85,B 0,C 180,E1 -10540.351,E2 -10540.351} C_VEL
LIN {X 0,Y 411.18,Z 513.389,A -85,B 0,C 180,E1 -10541.586,E2 -10541.586} C_VEL
LIN {X 0,Y 411.783,Z 503.508,A -85,B 0,C 180,E1 -10542.819,E2 -10542.819} C_VEL
LIN {X 0,Y 412.122,Z 495.252,A -85,B 0,C 180,E1 -10543.664,E2 -10543.664} C_VEL
LIN {X 0,Y 412.704,Z 484.76,A -85,B 0,C 180,E1 -10544.547,E2 -10544.547} C_VEL
LIN {X 0,Y 413.272,Z 472.428,A -85,B 0,C 180,E1 -10545.346,E2 -10545.346} C_VEL
LIN {X 0,Y 413.321,Z 466.46,A -85,B 0,C 180,E1 -10545.66,E2 -10545.66} C_VEL
LIN {X 0,Y 412.2,Z 453.573,A -85,B 0,C 180,E1 -10546.212,E2 -10546.212} C_VEL
LIN {X 0,Y 411.292,Z 443.512,A -85,B 0,C 180,E1 -10546.504,E2 -10546.504} C_VEL
LIN {X 0,Y 412.063,Z 430.236,A -85,B 0,C 180,E1 -10549.685,E2 -10549.685} C_VEL
LIN {X 0,Y 413.124,Z 416.455,A -85,B 0,C 180,E1 -10553.034,E2 -10553.034} C_VEL
LIN {X 0,Y 414.431,Z 402.65,A -85,B 0,C 180,E1 -10556.433,E2 -10556.433} C_VEL
LIN {X 0,Y 415.602,Z 390.998,A -85,B 0,C 180,E1 -10559.367,E2 -10559.367} C_VEL
LIN {X 0,Y 414.251,Z 383.443,A -85,B 0,C 180,E1 -10561.446,E2 -10561.446} C_VEL
LIN {X 0,Y 411.902,Z 372.455,A -85,B 0,C 180,E1 -10564.603,E2 -10564.603} C_VEL
LIN {X 0,Y 411.227,Z 369.262,A -85,B 0,C 180,E1 -10565.601,E2 -10565.601} C_VEL
LIN {X 0,Y 411.218,Z 369.261,A -85,B 0,C 180,E1 -10569.224,E2 -10569.224} C_VEL
LIN {X 0,Y 411.186,Z 369.266,A -85,B 0,C 180,E1 -10572.696,E2 -10572.696} C_VEL
LIN {X 0,Y 411.175,Z 369.268,A -85,B 0,C 180,E1 -10575.88,E2 -10575.88} C_VEL
LIN {X 0,Y 411.207,Z 369.262,A -85,B 0,C 180,E1 -10579.499,E2 -10579.499} C_VEL
LIN {X 0,Y 411.202,Z 369.267,A -85,B 0,C 180,E1 -10582.027,E2 -10582.027} C_VEL
LIN {X 0,Y 411.207,Z 369.265,A -85,B 0,C 180,E1 -10585.666,E2 -10585.666} C_VEL
LIN {X 0,Y 411.19,Z 369.264,A -85,B 0,C 180,E1 -10589.152,E2 -10589.152} C_VEL
LIN {X 0,Y 411.26,Z 369.256,A -85,B 0,C 180,E1 -10592.522,E2 -10592.522} C_VEL
LIN {X 0,Y 411.228,Z 369.262,A -85,B 0,C 180,E1 -10595.785,E2 -10595.785} C_VEL
LIN {X 0,Y 411.198,Z 369.263,A -85,B 0,C 180,E1 -10598.966,E2 -10598.966} C_VEL
LIN {X 0,Y 411.254,Z 369.258,A -85,B 0,C 180,E1 -10602.085,E2 -10602.085} C_VEL
LIN {X 0,Y 411.262,Z 369.256,A -85,B 0,C 180,E1 -10605.147,E2 -10605.147} C_VEL
LIN {X 0,Y 411.285,Z 369.255,A -85,B 0,C 180,E1 -10608.167,E2 -10608.167} C_VEL
LIN {X 0,Y 411.483,Z 369.228,A -85,B 0,C 180,E1 -10612.147,E2 -10612.147} C_VEL
LIN {X 0,Y 411.476,Z 369.229,A -85,B 0,C 180,E1 -10614.118,E2 -10614.118} C_VEL
LIN {X 0,Y 411.515,Z 369.226,A -85,B 0,C 180,E1 -10618.043,E2 -10618.043} C_VEL
LIN {X 0,Y 411.644,Z 369.21,A -85,B 0,C 180,E1 -10620,E2 -10620} C_VEL
LIN {X 0,Y 411.459,Z 369.231,A -85,B 0,C 180,E1 -10622.937,E2 -10622.937} C_VEL
LIN {X 0,Y 411.462,Z 369.232,A -85,B 0,C 180,E1 -10626.867,E2 -10626.867} C_VEL
LIN {X 0,Y 411.309,Z 369.252,A -85,B 0,C 180,E1 -10629.838,E2 -10629.838} C_VEL
LIN {X 0,Y 411.315,Z 369.251,A -85,B 0,C 180,E1 -10633.109,E2 -10633.109} C_VEL
LIN {X 0,Y 411.258,Z 369.258,A -85,B 0,C 180,E1 -10636.889,E2 -10636.889} C_VEL
LIN {X 0,Y 411.231,Z 369.26,A -85,B 0,C 180,E1 -10639.987,E2 -10639.987} C_VEL
LIN {X 0,Y 411.204,Z 369.265,A -85,B 0,C 180,E1 -10643.148,E2 -10643.148} C_VEL
LIN {X 0,Y 411.239,Z 369.257,A -85,B 0,C 180,E1 -10646.381,E2 -10646.381} C_VEL
LIN {X 0,Y 411.201,Z 369.264,A -85,B 0,C 180,E1 -10649.713,E2 -10649.713} C_VEL
LIN {X 0,Y 411.207,Z 369.265,A -85,B 0,C 180,E1 -10653.156,E2 -10653.156} C_VEL
LIN {X 0,Y 411.196,Z 369.265,A -85,B 0,C 180,E1 -10656.553,E2 -10656.553} C_VEL
LIN {X 0,Y 411.216,Z 369.261,A -85,B 0,C 180,E1 -10659.728,E2 -10659.728} C_VEL
LIN {X 0,Y 411.174,Z 369.269,A -85,B 0,C 180,E1 -10663.134,E2 -10663.134} C_VEL
LIN {X 0,Y 411.174,Z 369.266,A -85,B 0,C 180,E1 -10665.88,E2 -10665.88} C_VEL
LIN {X 0,Y 411.167,Z 369.271,A -85,B 0,C 180,E1 -10668.771,E2 -10668.771} C_VEL
LIN {X 0,Y 411.208,Z 369.262,A -85,B 0,C 180,E1 -10671.831,E2 -10671.831} C_VEL
